LIN {X 0,Y 296.903,Z 465.788,A -85,B 0,C 180,E1 -16297.482,E2 -16297.482} C_VEL
LIN {X 0,Y 297.504,Z 461.29,A -85,B 0,C 180,E1 -16299.52,E2 -16299.52} C_VEL
LIN {X 0,Y 298.387,Z 455.128,A -85,B 0,C 180,E1 -16301.55,E2 -16301.55} C_VEL
LIN {X 0,Y 299.207,Z 450.07,A -85,B 0,C 180,E1 -16302.895,E2 -16302.895} C_VEL
LIN {X 0,Y 300.204,Z 444.009,A -85,B 0,C 180,E1 -16304.232,E2 -16304.232} C_VEL
LIN {X 0,Y 301.376,Z 436.681,A -85,B 0,C 180,E1 -16305.557,E2 -16305.557} C_VEL
LIN {X 0,Y 302.09,Z 430.75,A -85,B 0,C 180,E1 -16306.471,E2 -16306.471} C_VEL
LIN {X 0,Y 302.187,Z 422.359,A -85,B 0,C 180,E1 -16307.6,E2 -16307.6} C_VEL
LIN {X 0,Y 301.805,Z 414.568,A -85,B 0,C 180,E1 -16308.5,E2 -16308.5} C_VEL
LIN {X 0,Y 300.734,Z 405.095,A -85,B 0,C 180,E1 -16309.432,E2 -16309.432} C_VEL
LIN {X 0,Y 298.864,Z 395.139,A -85,B 0,C 180,E1 -16310.262,E2 -16310.262} C_VEL
LIN {X 0,Y 297.662,Z 389.505,A -85,B 0,C 180,E1 -16310.689,E2 -16310.689} C_VEL
LIN {X 0,Y 298.446,Z 382.63,A -85,B 0,C 180,E1 -16315.081,E2 -16315.081} C_VEL
LIN {X 0,Y 299.306,Z 377.058,A -85,B 0,C 180,E1 -16318.776,E2 -16318.776} C_VEL
LIN {X 0,Y 300.359,Z 371.535,A -85,B 0,C 180,E1 -16322.609,E2 -16322.609} C_VEL
LIN {X 0,Y 300.474,Z 369.453,A -85,B 0,C 180,E1 -16324.151,E2 -16324.151} C_VEL
LIN {X 0,Y 300.035,Z 365.619,A -85,B 0,C 180,E1 -16327.21,E2 -16327.21} C_VEL
LIN {X 0,Y 299.34,Z 361.171,A -85,B 0,C 180,E1 -16331.103,E2 -16331.103} C_VEL
LIN {X 0,Y 298.551,Z 357.134,A -85,B 0,C 180,E1 -16335.071,E2 -16335.071} C_VEL
LIN {X 0,Y 298.382,Z 356.135,A -85,B 0,C 180,E1 -16336.22,E2 -16336.22} C_VEL
LIN {X 0,Y 298.411,Z 356.128,A -85,B 0,C 180,E1 -16340.513,E2 -16340.513} C_VEL
LIN {X 0,Y 298.427,Z 356.126,A -85,B 0,C 180,E1 -16343.93,E2 -16343.93} C_VEL
LIN {X 0,Y 298.402,Z 356.129,A -85,B 0,C 180,E1 -16347.984,E2 -16347.984} C_VEL
LIN {X 0,Y 298.467,Z 356.121,A -85,B 0,C 180,E1 -16351.904,E2 -16351.904} C_VEL
LIN {X 0,Y 298.494,Z 356.118,A -85,B 0,C 180,E1 -16354.924,E2 -16354.924} C_VEL
LIN {X 0,Y 298.459,Z 356.121,A -85,B 0,C 180,E1 -16359.315,E2 -16359.315} C_VEL
LIN {X 0,Y 298.546,Z 356.111,A -85,B 0,C 180,E1 -16362.179,E2 -16362.179} C_VEL
LIN {X 0,Y 298.602,Z 356.104,A -85,B 0,C 180,E1 -16364.994,E2 -16364.994} C_VEL
LIN {X 0,Y 298.591,Z 356.104,A -85,B 0,C 180,E1 -16369.145,E2 -16369.145} C_VEL
LIN {X 0,Y 298.72,Z 356.089,A -85,B 0,C 180,E1 -16371.884,E2 -16371.884} C_VEL
LIN {X 0,Y 298.646,Z 356.098,A -85,B 0,C 180,E1 -16374.597,E2 -16374.597} C_VEL
LIN {X 0,Y 298.928,Z 356.059,A -85,B 0,C 180,E1 -16378.652,E2 -16378.652} C_VEL
LIN {X 0,Y 298.928,Z 356.06,A -85,B 0,C 180,E1 -16381.346,E2 -16381.346} C_VEL
LIN {X 0,Y 298.781,Z 356.083,A -85,B 0,C 180,E1 -16386.753,E2 -16386.753} C_VEL
LIN {X 0,Y 298.631,Z 356.1,A -85,B 0,C 180,E1 -16389.481,E2 -16389.481} C_VEL
LIN {X 0,Y 298.544,Z 356.115,A -85,B 0,C 180,E1 -16393.614,E2 -16393.614} C_VEL
LIN {X 0,Y 298.527,Z 356.119,A -85,B 0,C 180,E1 -16395.148,E2 -16395.148} C_VEL
LIN {X 0,Y 298.42,Z 356.43,A -85,B 0,C 180,E1 -16396.414,E2 -16396.414} C_VEL
LIN {X 0,Y 298.385,Z 358.776,A -85,B 0,C 180,E1 -16399.582,E2 -16399.582} C_VEL
LIN {X 0,Y 298.025,Z 362.016,A -85,B 0,C 180,E1 -16403.632,E2 -16403.632} C_VEL
LIN {X 0,Y 297.777,Z 364.531,A -85,B 0,C 180,E1 -16406.641,E2 -16406.641} C_VEL
LIN {X 0,Y 297.563,Z 366.942,A -85,B 0,C 180,E1 -16409.443,E2 -16409.443} C_VEL
LIN {X 0,Y 301.042,Z 378.514,A -85,B 0,C 180,E1 -16410.513,E2 -16410.513} C_VEL
LIN {X 0,Y 303.065,Z 387.21,A -85,B 0,C 180,E1 -16411.449,E2 -16411.449} C_VEL
LIN {X 0,Y 304.331,Z 395.51,A -85,B 0,C 180,E1 -16412.468,E2 -16412.468} C_VEL
LIN {X 0,Y 304.232,Z 400.04,A -85,B 0,C 180,E1 -16413.028,E2 -16413.028} C_VEL
LIN {X 0,Y 303.064,Z 408.255,A -85,B 0,C 180,E1 -16414.191,E2 -16414.191} C_VEL
LIN {X 0,Y 301.948,Z 415.449,A -85,B 0,C 180,E1 -16415.446,E2 -16415.446} C_VEL
LIN {X 0,Y 300.854,Z 422.227,A -85,B 0,C 180,E1 -16416.897,E2 -16416.897} C_VEL
LIN {X 0,Y 299.851,Z 427.76,A -85,B 0,C 180,E1 -16418.344,E2 -16418.344} C_VEL
LIN {X 0,Y 299.089,Z 432.231,A -85,B 0,C 180,E1 -16419.778,E2 -16419.778} C_VEL
LIN {X 0,Y 298.316,Z 436.018,A -85,B 0,C 180,E1 -16421.271,E2 -16421.271} C_VEL
LIN {X 0,Y 297.7,Z 439.323,A -85,B 0,C 180,E1 -16422.957,E2 -16422.957} C_VEL
LIN {X 0,Y 297.154,Z 441.914,A -85,B 0,C 180,E1 -16424.801,E2 -16424.801} C_VEL
LIN {X 0,Y 296.657,Z 443.922,A -85,B 0,C 180,E1 -16427.255,E2 -16427.255} C_VEL
LIN {X 0,Y 296.462,Z 444.243,A -85,B 0,C 180,E1 -16429.338,E2 -16429.338} C_VEL
LIN {X 0,Y 296.511,Z 442.977,A -85,B 0,C 180,E1 -16431.955,E2 -16431.955} C_VEL
LIN {X 0,Y 296.695,Z 441.119,A -85,B 0,C 180,E1 -16433.686,E2 -16433.686} C_VEL
LIN {X 0,Y 297.078,Z 437.521,A -85,B 0,C 180,E1 -16435.89,E2 -16435.89} C_VEL
LIN {X 0,Y 297.534,Z 433.319,A -85,B 0,C 180,E1 -16437.684,E2 -16437.684} C_VEL
LIN {X 0,Y 298.153,Z 427.612,A -85,B 0,C 180,E1 -16439.548,E2 -16439.548} C_VEL
LIN {X 0,Y 298.758,Z 422.641,A -85,B 0,C 180,E1 -16440.866,E2 -16440.866} C_VEL
LIN {X 0,Y 299.406,Z 416.321,A -85,B 0,C 180,E1 -16442.255,E2 -16442.255} C_VEL
LIN {X 0,Y 300.027,Z 410.818,A -85,B 0,C 180,E1 -16443.274,E2 -16443.274} C_VEL
LIN {X 0,Y 300.724,Z 403.711,A -85,B 0,C 180,E1 -16444.382,E2 -16444.382} C_VEL
LIN {X 0,Y 301.459,Z 395.806,A -85,B 0,C 180,E1 -16445.393,E2 -16445.393} C_VEL
LIN {X 0,Y 301.683,Z 390.975,A -85,B 0,C 180,E1 -16445.939,E2 -16445.939} C_VEL
LIN {X 0,Y 300.083,Z 380.873,A -85,B 0,C 180,E1 -16446.933,E2 -16446.933} C_VEL
LIN {X 0,Y 298.191,Z 370.982,A -85,B 0,C 180,E1 -16447.696,E2 -16447.696} C_VEL
LIN {X 0,Y 297.089,Z 365.25,A -85,B 0,C 180,E1 -16448.078,E2 -16448.078} C_VEL
LIN {X 0,Y 297.245,Z 361.276,A -85,B 0,C 180,E1 -16452.098,E2 -16452.098} C_VEL
LIN {X 0,Y 297.576,Z 357.178,A -85,B 0,C 180,E1 -16456.337,E2 -16456.337} C_VEL
LIN {X 0,Y 297.68,Z 356.218,A -85,B 0,C 180,E1 -16457.73,E2 -16457.73} C_VEL
LIN {X 0,Y 298.506,Z 356.113,A -85,B 0,C 180,E1 -16461.877,E2 -16461.877} C_VEL
LIN {X 0,Y 298.621,Z 356.1,A -85,B 0,C 180,E1 -16464.597,E2 -16464.597} C_VEL
LIN {X 0,Y 298.916,Z 356.062,A -85,B 0,C 180,E1 -16468.651,E2 -16468.651} C_VEL
LIN {X 0,Y 298.914,Z 356.061,A -85,B 0,C 180,E1 -16471.346,E2 -16471.346} C_VEL
LIN {X 0,Y 298.789,Z 356.076,A -85,B 0,C 180,E1 -16476.752,E2 -16476.752} C_VEL
LIN {X 0,Y 298.67,Z 356.093,A -85,B 0,C 180,E1 -16479.479,E2 -16479.479} C_VEL
LIN {X 0,Y 298.542,Z 356.11,A -85,B 0,C 180,E1 -16483.614,E2 -16483.614} C_VEL
LIN {X 0,Y 298.537,Z 356.108,A -85,B 0,C 180,E1 -16486.407,E2 -16486.407} C_VEL
LIN {X 0,Y 298.499,Z 356.117,A -85,B 0,C 180,E1 -16489.653,E2 -16489.653} C_VEL
LIN {X 0,Y 298.445,Z 356.124,A -85,B 0,C 180,E1 -16493.597,E2 -16493.597} C_VEL
LIN {X 0,Y 298.476,Z 356.115,A -85,B 0,C 180,E1 -16496.573,E2 -16496.573} C_VEL
LIN {X 0,Y 298.407,Z 356.127,A -85,B 0,C 180,E1 -16499.64,E2 -16499.64} C_VEL
LIN {X 0,Y 298.382,Z 356.128,A -85,B 0,C 180,E1 -16502.799,E2 -16502.799} C_VEL
LIN {X 0,Y 298.458,Z 356.119,A -85,B 0,C 180,E1 -16506.814,E2 -16506.814} C_VEL
LIN {X 0,Y 298.443,Z 356.124,A -85,B 0,C 180,E1 -16511.103,E2 -16511.103} C_VEL
LIN {X 0,Y 298.475,Z 356.12,A -85,B 0,C 180,E1 -16515.061,E2 -16515.061} C_VEL
LIN {X 0,Y 298.443,Z 356.124,A -85,B 0,C 180,E1 -16518.897,E2 -16518.897} C_VEL
LIN {X 0,Y 298.457,Z 356.119,A -85,B 0,C 180,E1 -16523.186,E2 -16523.186} C_VEL
LIN {X 0,Y 298.382,Z 356.129,A -85,B 0,C 180,E1 -16527.2,E2 -16527.2} C_VEL
LIN {X 0,Y 298.418,Z 356.127,A -85,B 0,C 180,E1 -16530.615,E2 -16530.615} C_VEL
LIN {X 0,Y 298.472,Z 356.116,A -85,B 0,C 180,E1 -16533.474,E2 -16533.474} C_VEL
LIN {X 0,Y 298.507,Z 356.115,A -85,B 0,C 180,E1 -16536.66,E2 -16536.66} C_VEL
LIN {X 0,Y 298.554,Z 356.108,A -85,B 0,C 180,E1 -16540.759,E2 -16540.759} C_VEL
LIN {X 0,Y 298.581,Z 356.103,A -85,B 0,C 180,E1 -16544.996,E2 -16544.996} C_VEL
LIN {X 0,Y 298.583,Z 356.102,A -85,B 0,C 180,E1 -16549.148,E2 -16549.148} C_VEL
LIN {X 0,Y 298.747,Z 356.084,A -85,B 0,C 180,E1 -16551.887,E2 -16551.887} C_VEL
LIN {X 0,Y 298.65,Z 356.094,A -85,B 0,C 180,E1 -16554.6,E2 -16554.6} C_VEL
LIN {X 0,Y 298.828,Z 356.071,A -85,B 0,C 180,E1 -16557.415,E2 -16557.415} C_VEL
LIN {X 0,Y 298.194,Z 356.152,A -85,B 0,C 180,E1 -16558.541,E2 -16558.541} C_VEL
LIN {X 0,Y 295.394,Z 356.501,A -85,B 0,C 180,E1 -16560.377,E2 -16560.377} C_VEL
LIN {X 0,Y 292.07,Z 356.914,A -85,B 0,C 180,E1 -16562.628,E2 -16562.628} C_VEL
LIN {X 0,Y 291.651,Z 356.963,A -85,B 0,C 180,E1 -16563.408,E2 -16563.408} C_VEL
LIN {X 0,Y 291.736,Z 356.955,A -85,B 0,C 180,E1 -16566.919,E2 -16566.919} C_VEL
LIN {X 0,Y 291.62,Z 356.974,A -85,B 0,C 180,E1 -16569.713,E2 -16569.713} C_VEL
LIN {X 0,Y 291.514,Z 356.985,A -85,B 0,C 180,E1 -16573.952,E2 -16573.952} C_VEL
LIN {X 0,Y 291.478,Z 356.987,A -85,B 0,C 180,E1 -16576.82,E2 -16576.82} C_VEL
LIN {X 0,Y 291.442,Z 356.992,A -85,B 0,C 180,E1 -16579.877,E2 -16579.877} C_VEL
LIN {X 0,Y 291.392,Z 356.998,A -85,B 0,C 180,E1 -16584.207,E2 -16584.207} C_VEL
LIN {X 0,Y 291.416,Z 357,A -85,B 0,C 180,E1 -16587.273,E2 -16587.273} C_VEL
LIN {X 0,Y 291.331,Z 357.005,A -85,B 0,C 180,E1 -16590.439,E2 -16590.439} C_VEL
LIN {X 0,Y 291.338,Z 357.005,A -85,B 0,C 180,E1 -16593.7,E2 -16593.7} C_VEL
LIN {X 0,Y 291.367,Z 357.004,A -85,B 0,C 180,E1 -16597.255,E2 -16597.255} C_VEL
LIN {X 0,Y 291.327,Z 357.008,A -85,B 0,C 180,E1 -16600.645,E2 -16600.645} C_VEL
LIN {X 0,Y 291.309,Z 357.009,A -85,B 0,C 180,E1 -16604.399,E2 -16604.399} C_VEL
LIN {X 0,Y 291.415,Z 357.077,A -85,B 0,C 180,E1 -16608.646,E2 -16608.646} C_VEL
LIN {X 0,Y 292.375,Z 362.103,A -85,B 0,C 180,E1 -16612.491,E2 -16612.491} C_VEL
LIN {X 0,Y 292.972,Z 366.53,A -85,B 0,C 180,E1 -16615.688,E2 -16615.688} C_VEL
LIN {X 0,Y 292.883,Z 368.616,A -85,B 0,C 180,E1 -16617.126,E2 -16617.126} C_VEL
LIN {X 0,Y 292.227,Z 372.868,A -85,B 0,C 180,E1 -16619.975,E2 -16619.975} C_VEL
LIN {X 0,Y 291.277,Z 379.444,A -85,B 0,C 180,E1 -16624.261,E2 -16624.261} C_VEL
LIN {X 0,Y 290.503,Z 386.389,A -85,B 0,C 180,E1 -16628.724,E2 -16628.724} C_VEL
LIN {X 0,Y 290.108,Z 390.872,A -85,B 0,C 180,E1 -16631.559,E2 -16631.559} C_VEL
LIN {X 0,Y 291.601,Z 403.954,A -85,B 0,C 180,E1 -16632.378,E2 -16632.378} C_VEL
LIN {X 0,Y 292.484,Z 413.89,A -85,B 0,C 180,E1 -16633.243,E2 -16633.243} C_VEL
LIN {X 0,Y 293.002,Z 422.205,A -85,B 0,C 180,E1 -16634.146,E2 -16634.146} C_VEL
LIN {X 0,Y 293.138,Z 429.314,A -85,B 0,C 180,E1 -16635.066,E2 -16635.066} C_VEL
LIN {X 0,Y 292.254,Z 437.158,A -85,B 0,C 180,E1 -16636.265,E2 -16636.265} C_VEL
LIN {X 0,Y 291.523,Z 443.666,A -85,B 0,C 180,E1 -16637.471,E2 -16637.471} C_VEL
LIN {X 0,Y 290.863,Z 449.871,A -85,B 0,C 180,E1 -16638.856,E2 -16638.856} C_VEL
LIN {X 0,Y 290.376,Z 455.026,A -85,B 0,C 180,E1 -16640.248,E2 -16640.248} C_VEL
LIN {X 0,Y 289.995,Z 459.311,A -85,B 0,C 180,E1 -16641.641,E2 -16641.641} C_VEL
LIN {X 0,Y 289.715,Z 462.857,A -85,B 0,C 180,E1 -16643.035,E2 -16643.035} C_VEL
LIN {X 0,Y 289.532,Z 466.528,A -85,B 0,C 180,E1 -16644.896,E2 -16644.896} C_VEL
LIN {X 0,Y 289.575,Z 468.046,A -85,B 0,C 180,E1 -16645.826,E2 -16645.826} C_VEL
LIN {X 0,Y 289.545,Z 469.683,A -85,B 0,C 180,E1 -16647.219,E2 -16647.219} C_VEL
LIN {X 0,Y 289.531,Z 470.791,A -85,B 0,C 180,E1 -16648.611,E2 -16648.611} C_VEL
LIN {X 0,Y 289.582,Z 471.416,A -85,B 0,C 180,E1 -16650.002,E2 -16650.002} C_VEL
LIN {X 0,Y 289.514,Z 471.562,A -85,B 0,C 180,E1 -16651.393,E2 -16651.393} C_VEL
LIN {X 0,Y 289.519,Z 471.172,A -85,B 0,C 180,E1 -16652.785,E2 -16652.785} C_VEL
LIN {X 0,Y 289.505,Z 470.202,A -85,B 0,C 180,E1 -16654.178,E2 -16654.178} C_VEL
LIN {X 0,Y 289.52,Z 468.751,A -85,B 0,C 180,E1 -16655.574,E2 -16655.574} C_VEL
LIN {X 0,Y 289.855,Z 465.607,A -85,B 0,C 180,E1 -16657.665,E2 -16657.665} C_VEL
LIN {X 0,Y 290.472,Z 461.182,A -85,B 0,C 180,E1 -16659.753,E2 -16659.753} C_VEL
LIN {X 0,Y 291.415,Z 455.106,A -85,B 0,C 180,E1 -16661.831,E2 -16661.831} C_VEL
LIN {X 0,Y 292.292,Z 450.124,A -85,B 0,C 180,E1 -16663.206,E2 -16663.206} C_VEL
LIN {X 0,Y 293.333,Z 444.163,A -85,B 0,C 180,E1 -16664.572,E2 -16664.572} C_VEL
LIN {X 0,Y 294.566,Z 436.956,A -85,B 0,C 180,E1 -16665.927,E2 -16665.927} C_VEL
LIN {X 0,Y 295.338,Z 429.614,A -85,B 0,C 180,E1 -16667.089,E2 -16667.089} C_VEL
LIN {X 0,Y 295.352,Z 421.521,A -85,B 0,C 180,E1 -16668.2,E2 -16668.2} C_VEL
LIN {X 0,Y 294.915,Z 413.637,A -85,B 0,C 180,E1 -16669.129,E2 -16669.129} C_VEL
LIN {X 0,Y 293.8,Z 404.622,A -85,B 0,C 180,E1 -16670.045,E2 -16670.045} C_VEL
LIN {X 0,Y 291.838,Z 394.392,A -85,B 0,C 180,E1 -16670.93,E2 -16670.93} C_VEL
LIN {X 0,Y 290.722,Z 389.114,A -85,B 0,C 180,E1 -16671.355,E2 -16671.355} C_VEL
LIN {X 0,Y 291.518,Z 382.516,A -85,B 0,C 180,E1 -16675.72,E2 -16675.72} C_VEL
LIN {X 0,Y 292.266,Z 378.081,A -85,B 0,C 180,E1 -16678.748,E2 -16678.748} C_VEL
LIN {X 0,Y 293.441,Z 372.083,A -85,B 0,C 180,E1 -16683.042,E2 -16683.042} C_VEL
LIN {X 0,Y 293.376,Z 368.98,A -85,B 0,C 180,E1 -16685.462,E2 -16685.462} C_VEL
LIN {X 0,Y 292.834,Z 365.286,A -85,B 0,C 180,E1 -16688.611,E2 -16688.611} C_VEL
LIN {X 0,Y 292.107,Z 361.274,A -85,B 0,C 180,E1 -16692.353,E2 -16692.353} C_VEL
LIN {X 0,Y 291.383,Z 357.005,A -85,B 0,C 180,E1 -16696.931,E2 -16696.931} C_VEL
LIN {X 0,Y 291.361,Z 357.005,A -85,B 0,C 180,E1 -16701.158,E2 -16701.158} C_VEL
LIN {X 0,Y 291.37,Z 357.004,A -85,B 0,C 180,E1 -16704.626,E2 -16704.626} C_VEL
LIN {X 0,Y 291.379,Z 357.004,A -85,B 0,C 180,E1 -16707.95,E2 -16707.95} C_VEL
LIN {X 0,Y 291.386,Z 357.001,A -85,B 0,C 180,E1 -16711.158,E2 -16711.158} C_VEL
LIN {X 0,Y 291.423,Z 356.998,A -85,B 0,C 180,E1 -16714.271,E2 -16714.271} C_VEL
LIN {X 0,Y 291.39,Z 357.001,A -85,B 0,C 180,E1 -16717.299,E2 -16717.299} C_VEL
LIN {X 0,Y 291.467,Z 356.992,A -85,B 0,C 180,E1 -16720.27,E2 -16720.27} C_VEL
LIN {X 0,Y 291.564,Z 356.98,A -85,B 0,C 180,E1 -16724.623,E2 -16724.623} C_VEL
LIN {X 0,Y 291.537,Z 356.983,A -85,B 0,C 180,E1 -16728.879,E2 -16728.879} C_VEL
LIN {X 0,Y 291.671,Z 356.968,A -85,B 0,C 180,E1 -16731.686,E2 -16731.686} C_VEL
LIN {X 0,Y 291.615,Z 356.974,A -85,B 0,C 180,E1 -16734.467,E2 -16734.467} C_VEL
LIN {X 0,Y 291.894,Z 356.935,A -85,B 0,C 180,E1 -16738.619,E2 -16738.619} C_VEL
LIN {X 0,Y 291.894,Z 356.936,A -85,B 0,C 180,E1 -16741.378,E2 -16741.378} C_VEL
LIN {X 0,Y 291.729,Z 356.96,A -85,B 0,C 180,E1 -16746.917,E2 -16746.917} C_VEL
LIN {X 0,Y 291.573,Z 356.98,A -85,B 0,C 180,E1 -16749.712,E2 -16749.712} C_VEL
LIN {X 0,Y 291.504,Z 356.991,A -85,B 0,C 180,E1 -16753.95,E2 -16753.95} C_VEL
LIN {X 0,Y 291.462,Z 357,A -85,B 0,C 180,E1 -16755.38,E2 -16755.38} C_VEL
LIN {X 0,Y 291.416,Z 358.946,A -85,B 0,C 180,E1 -16758.27,E2 -16758.27} C_VEL
LIN {X 0,Y 291.187,Z 361.179,A -85,B 0,C 180,E1 -16761.224,E2 -16761.224} C_VEL
LIN {X 0,Y 290.947,Z 363.568,A -85,B 0,C 180,E1 -16764.244,E2 -16764.244} C_VEL
LIN {X 0,Y 290.611,Z 366.768,A -85,B 0,C 180,E1 -16768.135,E2 -16768.135} C_VEL
LIN {X 0,Y 290.552,Z 367.318,A -85,B 0,C 180,E1 -16768.782,E2 -16768.782} C_VEL
LIN {X 0,Y 293.885,Z 378.073,A -85,B 0,C 180,E1 -16769.815,E2 -16769.815} C_VEL
LIN {X 0,Y 296.191,Z 387.481,A -85,B 0,C 180,E1 -16770.87,E2 -16770.87} C_VEL
LIN {X 0,Y 297.513,Z 395.491,A -85,B 0,C 180,E1 -16771.885,E2 -16771.885} C_VEL
LIN {X 0,Y 297.828,Z 398.291,A -85,B 0,C 180,E1 -16772.266,E2 -16772.266} C_VEL
LIN {X 0,Y 296.435,Z 408.512,A -85,B 0,C 180,E1 -16773.698,E2 -16773.698} C_VEL
LIN {X 0,Y 295.162,Z 416.165,A -85,B 0,C 180,E1 -16775.067,E2 -16775.067} C_VEL
LIN {X 0,Y 294.199,Z 421.9,A -85,B 0,C 180,E1 -16776.313,E2 -16776.313} C_VEL
LIN {X 0,Y 293.202,Z 427.288,A -85,B 0,C 180,E1 -16777.718,E2 -16777.718} C_VEL
LIN {X 0,Y 292.372,Z 431.815,A -85,B 0,C 180,E1 -16779.152,E2 -16779.152} C_VEL
LIN {X 0,Y 291.546,Z 435.598,A -85,B 0,C 180,E1 -16780.604,E2 -16780.604} C_VEL
LIN {X 0,Y 290.764,Z 439.505,A -85,B 0,C 180,E1 -16782.59,E2 -16782.59} C_VEL
LIN {X 0,Y 290.124,Z 442.311,A -85,B 0,C 180,E1 -16784.625,E2 -16784.625} C_VEL
LIN {X 0,Y 289.654,Z 444.03,A -85,B 0,C 180,E1 -16786.708,E2 -16786.708} C_VEL
LIN {X 0,Y 289.396,Z 444.627,A -85,B 0,C 180,E1 -16789.026,E2 -16789.026} C_VEL
LIN {X 0,Y 289.349,Z 443.972,A -85,B 0,C 180,E1 -16791.006,E2 -16791.006} C_VEL
LIN {X 0,Y 289.532,Z 441.999,A -85,B 0,C 180,E1 -16793.225,E2 -16793.225} C_VEL
LIN {X 0,Y 289.721,Z 440.504,A -85,B 0,C 180,E1 -16794.394,E2 -16794.394} C_VEL
LIN {X 0,Y 290.047,Z 437.442,A -85,B 0,C 180,E1 -16796.129,E2 -16796.129} C_VEL
LIN {X 0,Y 290.497,Z 433.412,A -85,B 0,C 180,E1 -16797.857,E2 -16797.857} C_VEL
LIN {X 0,Y 291.053,Z 428.46,A -85,B 0,C 180,E1 -16799.529,E2 -16799.529} C_VEL
LIN {X 0,Y 291.786,Z 422.266,A -85,B 0,C 180,E1 -16801.2,E2 -16801.2} C_VEL
LIN {X 0,Y 292.375,Z 416.814,A -85,B 0,C 180,E1 -16802.418,E2 -16802.418} C_VEL
LIN {X 0,Y 293.146,Z 410.103,A -85,B 0,C 180,E1 -16803.669,E2 -16803.669} C_VEL
LIN {X 0,Y 293.944,Z 402.126,A -85,B 0,C 180,E1 -16804.894,E2 -16804.894} C_VEL
LIN {X 0,Y 294.697,Z 393.776,A -85,B 0,C 180,E1 -16805.933,E2 -16805.933} C_VEL
LIN {X 0,Y 294.368,Z 389.435,A -85,B 0,C 180,E1 -16806.426,E2 -16806.426} C_VEL
LIN {X 0,Y 293.048,Z 381.18,A -85,B 0,C 180,E1 -16807.248,E2 -16807.248} C_VEL
LIN {X 0,Y 291.154,Z 371.388,A -85,B 0,C 180,E1 -16808.027,E2 -16808.027} C_VEL
LIN {X 0,Y 290.004,Z 365.538,A -85,B 0,C 180,E1 -16808.449,E2 -16808.449} C_VEL
LIN {X 0,Y 290.162,Z 362.436,A -85,B 0,C 180,E1 -16811.645,E2 -16811.645} C_VEL
LIN {X 0,Y 290.48,Z 358.307,A -85,B 0,C 180,E1 -16815.997,E2 -16815.997} C_VEL
LIN {X 0,Y 290.577,Z 357.104,A -85,B 0,C 180,E1 -16817.426,E2 -16817.426} C_VEL
LIN {X 0,Y 291.442,Z 356.992,A -85,B 0,C 180,E1 -16821.679,E2 -16821.679} C_VEL
LIN {X 0,Y 291.585,Z 356.978,A -85,B 0,C 180,E1 -16824.466,E2 -16824.466} C_VEL
LIN {X 0,Y 291.882,Z 356.939,A -85,B 0,C 180,E1 -16828.619,E2 -16828.619} C_VEL
LIN {X 0,Y 291.88,Z 356.938,A -85,B 0,C 180,E1 -16831.378,E2 -16831.378} C_VEL
LIN {X 0,Y 291.738,Z 356.955,A -85,B 0,C 180,E1 -16836.916,E2 -16836.916} C_VEL
LIN {X 0,Y 291.619,Z 356.973,A -85,B 0,C 180,E1 -16839.71,E2 -16839.71} C_VEL
LIN {X 0,Y 291.511,Z 356.987,A -85,B 0,C 180,E1 -16843.949,E2 -16843.949} C_VEL
LIN {X 0,Y 291.475,Z 356.987,A -85,B 0,C 180,E1 -16846.817,E2 -16846.817} C_VEL
LIN {X 0,Y 291.438,Z 356.994,A -85,B 0,C 180,E1 -16849.874,E2 -16849.874} C_VEL
LIN {X 0,Y 291.387,Z 356.999,A -85,B 0,C 180,E1 -16854.204,E2 -16854.204} C_VEL
LIN {X 0,Y 291.41,Z 356.999,A -85,B 0,C 180,E1 -16857.271,E2 -16857.271} C_VEL
LIN {X 0,Y 291.324,Z 357.006,A -85,B 0,C 180,E1 -16860.436,E2 -16860.436} C_VEL
LIN {X 0,Y 291.331,Z 357.007,A -85,B 0,C 180,E1 -16863.698,E2 -16863.698} C_VEL
LIN {X 0,Y 291.393,Z 357.002,A -85,B 0,C 180,E1 -16867.261,E2 -16867.261} C_VEL
LIN {X 0,Y 291.393,Z 356.999,A -85,B 0,C 180,E1 -16870.63,E2 -16870.63} C_VEL
LIN {X 0,Y 291.393,Z 356.997,A -85,B 0,C 180,E1 -16874.379,E2 -16874.379} C_VEL
LIN {X 0,Y 291.377,Z 357.001,A -85,B 0,C 180,E1 -16878.39,E2 -16878.39} C_VEL
LIN {X 0,Y 291.374,Z 357.002,A -85,B 0,C 180,E1 -16881.164,E2 -16881.164} C_VEL
LIN {X 0,Y 291.372,Z 357.003,A -85,B 0,C 180,E1 -16884.63,E2 -16884.63} C_VEL
LIN {X 0,Y 291.358,Z 357.002,A -85,B 0,C 180,E1 -16887.951,E2 -16887.951} C_VEL
LIN {X 0,Y 291.369,Z 357.001,A -85,B 0,C 180,E1 -16891.159,E2 -16891.159} C_VEL
LIN {X 0,Y 291.412,Z 356.998,A -85,B 0,C 180,E1 -16894.273,E2 -16894.273} C_VEL
LIN {X 0,Y 291.434,Z 356.992,A -85,B 0,C 180,E1 -16897.306,E2 -16897.306} C_VEL
LIN {X 0,Y 291.501,Z 356.987,A -85,B 0,C 180,E1 -16900.275,E2 -16900.275} C_VEL
LIN {X 0,Y 291.543,Z 356.981,A -85,B 0,C 180,E1 -16904.625,E2 -16904.625} C_VEL
LIN {X 0,Y 291.526,Z 356.981,A -85,B 0,C 180,E1 -16908.882,E2 -16908.882} C_VEL
LIN {X 0,Y 291.697,Z 356.961,A -85,B 0,C 180,E1 -16911.69,E2 -16911.69} C_VEL
LIN {X 0,Y 291.62,Z 356.971,A -85,B 0,C 180,E1 -16914.47,E2 -16914.47} C_VEL
LIN {X 0,Y 291.879,Z 356.938,A -85,B 0,C 180,E1 -16918.622,E2 -16918.622} C_VEL
LIN {X 0,Y 291.881,Z 356.938,A -85,B 0,C 180,E1 -16921.381,E2 -16921.381} C_VEL
LIN {X 0,Y 291.651,Z 356.963,A -85,B 0,C 180,E1 -16923.408,E2 -16923.408} C_VEL
LIN {X 0,Y 290.879,Z 357.062,A -85,B 0,C 180,E1 -16924.56,E2 -16924.56} C_VEL
LIN {X 0,Y 288.083,Z 357.41,A -85,B 0,C 180,E1 -16926.441,E2 -16926.441} C_VEL
LIN {X 0,Y 284.953,Z 357.801,A -85,B 0,C 180,E1 -16928.75,E2 -16928.75} C_VEL
LIN {X 0,Y 284.594,Z 357.845,A -85,B 0,C 180,E1 -16929.546,E2 -16929.546} C_VEL
LIN {X 0,Y 284.473,Z 357.86,A -85,B 0,C 180,E1 -16934.304,E2 -16934.304} C_VEL
LIN {X 0,Y 284.417,Z 357.869,A -85,B 0,C 180,E1 -16937.25,E2 -16937.25} C_VEL
LIN {X 0,Y 284.371,Z 357.872,A -85,B 0,C 180,E1 -16940.244,E2 -16940.244} C_VEL
LIN {X 0,Y 284.362,Z 357.875,A -85,B 0,C 180,E1 -16943.877,E2 -16943.877} C_VEL
LIN {X 0,Y 284.39,Z 357.874,A -85,B 0,C 180,E1 -16947.176,E2 -16947.176} C_VEL
LIN {X 0,Y 284.289,Z 357.887,A -85,B 0,C 180,E1 -16951.276,E2 -16951.276} C_VEL
LIN {X 0,Y 284.335,Z 357.879,A -85,B 0,C 180,E1 -16955.35,E2 -16955.35} C_VEL
LIN {X 0,Y 284.303,Z 357.88,A -85,B 0,C 180,E1 -16958.172,E2 -16958.172} C_VEL
LIN {X 0,Y 284.264,Z 357.886,A -85,B 0,C 180,E1 -16962.127,E2 -16962.127} C_VEL
LIN {X 0,Y 284.281,Z 357.884,A -85,B 0,C 180,E1 -16966.197,E2 -16966.197} C_VEL
LIN {X 0,Y 284.358,Z 358.006,A -85,B 0,C 180,E1 -16968.495,E2 -16968.495} C_VEL
LIN {X 0,Y 285.216,Z 362.531,A -85,B 0,C 180,E1 -16972.048,E2 -16972.048} C_VEL
LIN {X 0,Y 285.935,Z 367.27,A -85,B 0,C 180,E1 -16975.578,E2 -16975.578} C_VEL
LIN {X 0,Y 285.807,Z 369.643,A -85,B 0,C 180,E1 -16977.252,E2 -16977.252} C_VEL
LIN {X 0,Y 284.854,Z 375.483,A -85,B 0,C 180,E1 -16981.244,E2 -16981.244} C_VEL
LIN {X 0,Y 283.99,Z 381.297,A -85,B 0,C 180,E1 -16985.123,E2 -16985.123} C_VEL
LIN {X 0,Y 283.387,Z 387.087,A -85,B 0,C 180,E1 -16988.927,E2 -16988.927} C_VEL
LIN {X 0,Y 283.079,Z 390.547,A -85,B 0,C 180,E1 -16991.173,E2 -16991.173} C_VEL
LIN {X 0,Y 284.541,Z 403.382,A -85,B 0,C 180,E1 -16992.019,E2 -16992.019} C_VEL
LIN {X 0,Y 285.359,Z 412.423,A -85,B 0,C 180,E1 -16992.812,E2 -16992.812} C_VEL
LIN {X 0,Y 285.914,Z 421.408,A -85,B 0,C 180,E1 -16993.796,E2 -16993.796} C_VEL
LIN {X 0,Y 286.114,Z 429.484,A -85,B 0,C 180,E1 -16994.873,E2 -16994.873} C_VEL
LIN {X 0,Y 285.214,Z 437.244,A -85,B 0,C 180,E1 -16996.101,E2 -16996.101} C_VEL
LIN {X 0,Y 284.374,Z 444.536,A -85,B 0,C 180,E1 -16997.513,E2 -16997.513} C_VEL
LIN {X 0,Y 283.586,Z 451.945,A -85,B 0,C 180,E1 -16999.29,E2 -16999.29} C_VEL
LIN {X 0,Y 283.032,Z 457.734,A -85,B 0,C 180,E1 -17001.074,E2 -17001.074} C_VEL
LIN {X 0,Y 282.662,Z 462.301,A -85,B 0,C 180,E1 -17002.861,E2 -17002.861} C_VEL
LIN {X 0,Y 282.439,Z 466.367,A -85,B 0,C 180,E1 -17004.98,E2 -17004.98} C_VEL
LIN {X 0,Y 282.489,Z 467.559,A -85,B 0,C 180,E1 -17005.722,E2 -17005.722} C_VEL
LIN {X 0,Y 282.473,Z 469.231,A -85,B 0,C 180,E1 -17007.15,E2 -17007.15} C_VEL
LIN {X 0,Y 282.449,Z 470.386,A -85,B 0,C 180,E1 -17008.576,E2 -17008.576} C_VEL
LIN {X 0,Y 282.495,Z 471.056,A -85,B 0,C 180,E1 -17010.002,E2 -17010.002} C_VEL
LIN {X 0,Y 282.433,Z 471.245,A -85,B 0,C 180,E1 -17011.428,E2 -17011.428} C_VEL
LIN {X 0,Y 282.445,Z 470.86,A -85,B 0,C 180,E1 -17012.854,E2 -17012.854} C_VEL
LIN {X 0,Y 282.422,Z 468.781,A -85,B 0,C 180,E1 -17015.497,E2 -17015.497} C_VEL
LIN {X 0,Y 282.793,Z 465.431,A -85,B 0,C 180,E1 -17017.858,E2 -17017.858} C_VEL
LIN {X 0,Y 283.456,Z 461.083,A -85,B 0,C 180,E1 -17019.997,E2 -17019.997} C_VEL
LIN {X 0,Y 284.466,Z 455.139,A -85,B 0,C 180,E1 -17022.124,E2 -17022.124} C_VEL
LIN {X 0,Y 285.589,Z 448.814,A -85,B 0,C 180,E1 -17023.884,E2 -17023.884} C_VEL
LIN {X 0,Y 286.73,Z 442.665,A -85,B 0,C 180,E1 -17025.279,E2 -17025.279} C_VEL
LIN {X 0,Y 287.91,Z 436.25,A -85,B 0,C 180,E1 -17026.487,E2 -17026.487} C_VEL
LIN {X 0,Y 288.546,Z 430.243,A -85,B 0,C 180,E1 -17027.475,E2 -17027.475} C_VEL
LIN {X 0,Y 288.615,Z 422.127,A -85,B 0,C 180,E1 -17028.641,E2 -17028.641} C_VEL
LIN {X 0,Y 288.211,Z 414.483,A -85,B 0,C 180,E1 -17029.592,E2 -17029.592} C_VEL
LIN {X 0,Y 287.182,Z 405.595,A -85,B 0,C 180,E1 -17030.554,E2 -17030.554} C_VEL
LIN {X 0,Y 285.362,Z 395.938,A -85,B 0,C 180,E1 -17031.455,E2 -17031.455} C_VEL
LIN {X 0,Y 283.763,Z 388.785,A -85,B 0,C 180,E1 -17032.049,E2 -17032.049} C_VEL
LIN {X 0,Y 284.604,Z 382.426,A -85,B 0,C 180,E1 -17036.393,E2 -17036.393} C_VEL
LIN {X 0,Y 285.676,Z 376.57,A -85,B 0,C 180,E1 -17040.564,E2 -17040.564} C_VEL
LIN {X 0,Y 286.543,Z 372.636,A -85,B 0,C 180,E1 -17043.496,E2 -17043.496} C_VEL
LIN {X 0,Y 286.115,Z 368.434,A -85,B 0,C 180,E1 -17047.001,E2 -17047.001} C_VEL
LIN {X 0,Y 285.563,Z 364.845,A -85,B 0,C 180,E1 -17050.274,E2 -17050.274} C_VEL
LIN {X 0,Y 284.819,Z 360.852,A -85,B 0,C 180,E1 -17054.308,E2 -17054.308} C_VEL
LIN {X 0,Y 284.305,Z 357.886,A -85,B 0,C 180,E1 -17057.773,E2 -17057.773} C_VEL
LIN {X 0,Y 284.32,Z 357.883,A -85,B 0,C 180,E1 -17061.831,E2 -17061.831} C_VEL
LIN {X 0,Y 284.317,Z 357.883,A -85,B 0,C 180,E1 -17065.351,E2 -17065.351} C_VEL
LIN {X 0,Y 284.302,Z 357.885,A -85,B 0,C 180,E1 -17068.725,E2 -17068.725} C_VEL
LIN {X 0,Y 284.404,Z 357.872,A -85,B 0,C 180,E1 -17072.827,E2 -17072.827} C_VEL
LIN {X 0,Y 284.375,Z 357.875,A -85,B 0,C 180,E1 -17076.707,E2 -17076.707} C_VEL
LIN {X 0,Y 284.412,Z 357.87,A -85,B 0,C 180,E1 -17081.261,E2 -17081.261} C_VEL
LIN {X 0,Y 284.501,Z 357.859,A -85,B 0,C 180,E1 -17084.458,E2 -17084.458} C_VEL
LIN {X 0,Y 284.49,Z 357.861,A -85,B 0,C 180,E1 -17088.6,E2 -17088.6} C_VEL
LIN {X 0,Y 284.626,Z 357.845,A -85,B 0,C 180,E1 -17091.479,E2 -17091.479} C_VEL
LIN {X 0,Y 284.585,Z 357.851,A -85,B 0,C 180,E1 -17094.33,E2 -17094.33} C_VEL
LIN {X 0,Y 284.86,Z 357.811,A -85,B 0,C 180,E1 -17098.585,E2 -17098.585} C_VEL
LIN {X 0,Y 284.861,Z 357.812,A -85,B 0,C 180,E1 -17101.412,E2 -17101.412} C_VEL
LIN {X 0,Y 284.679,Z 357.838,A -85,B 0,C 180,E1 -17107.089,E2 -17107.089} C_VEL
LIN {X 0,Y 284.519,Z 357.859,A -85,B 0,C 180,E1 -17109.955,E2 -17109.955} C_VEL
LIN {X 0,Y 284.451,Z 357.871,A -85,B 0,C 180,E1 -17114.303,E2 -17114.303} C_VEL
LIN {X 0,Y 284.446,Z 358.391,A -85,B 0,C 180,E1 -17115.769,E2 -17115.769} C_VEL
LIN {X 0,Y 284.306,Z 361.404,A -85,B 0,C 180,E1 -17120.053,E2 -17120.053} C_VEL
LIN {X 0,Y 283.972,Z 364.195,A -85,B 0,C 180,E1 -17123.69,E2 -17123.69} C_VEL
LIN {X 0,Y 283.621,Z 367.44,A -85,B 0,C 180,E1 -17127.751,E2 -17127.751} C_VEL
LIN {X 0,Y 283.599,Z 367.847,A -85,B 0,C 180,E1 -17128.087,E2 -17128.087} C_VEL
LIN {X 0,Y 287.32,Z 379.582,A -85,B 0,C 180,E1 -17129.287,E2 -17129.287} C_VEL
LIN {X 0,Y 289.451,Z 388.306,A -85,B 0,C 180,E1 -17130.319,E2 -17130.319} C_VEL
LIN {X 0,Y 290.739,Z 395.754,A -85,B 0,C 180,E1 -17131.311,E2 -17131.311} C_VEL
LIN {X 0,Y 290.968,Z 401.422,A -85,B 0,C 180,E1 -17132.097,E2 -17132.097} C_VEL
LIN {X 0,Y 289.562,Z 410.212,A -85,B 0,C 180,E1 -17133.43,E2 -17133.43} C_VEL
LIN {X 0,Y 288.347,Z 417.223,A -85,B 0,C 180,E1 -17134.745,E2 -17134.745} C_VEL
LIN {X 0,Y 287.218,Z 423.361,A -85,B 0,C 180,E1 -17136.147,E2 -17136.147} C_VEL
LIN {X 0,Y 286.21,Z 428.471,A -85,B 0,C 180,E1 -17137.559,E2 -17137.559} C_VEL
LIN {X 0,Y 285.335,Z 432.971,A -85,B 0,C 180,E1 -17139.075,E2 -17139.075} C_VEL
LIN {X 0,Y 284.49,Z 436.591,A -85,B 0,C 180,E1 -17140.566,E2 -17140.566} C_VEL
LIN {X 0,Y 283.886,Z 439.452,A -85,B 0,C 180,E1 -17142.037,E2 -17142.037} C_VEL
LIN {X 0,Y 283.213,Z 442.252,A -85,B 0,C 180,E1 -17144.011,E2 -17144.011} C_VEL
LIN {X 0,Y 282.683,Z 444.127,A -85,B 0,C 180,E1 -17146.134,E2 -17146.134} C_VEL
LIN {X 0,Y 282.349,Z 444.91,A -85,B 0,C 180,E1 -17148.306,E2 -17148.306} C_VEL
LIN {X 0,Y 282.268,Z 444.545,A -85,B 0,C 180,E1 -17150.517,E2 -17150.517} C_VEL
LIN {X 0,Y 282.468,Z 442.184,A -85,B 0,C 180,E1 -17153.333,E2 -17153.333} C_VEL
LIN {X 0,Y 282.73,Z 439.639,A -85,B 0,C 180,E1 -17155.128,E2 -17155.128} C_VEL
LIN {X 0,Y 283.162,Z 436.204,A -85,B 0,C 180,E1 -17156.903,E2 -17156.903} C_VEL
LIN {X 0,Y 283.762,Z 430.876,A -85,B 0,C 180,E1 -17159.001,E2 -17159.001} C_VEL
LIN {X 0,Y 284.505,Z 424.924,A -85,B 0,C 180,E1 -17160.797,E2 -17160.797} C_VEL
LIN {X 0,Y 285.34,Z 417.34,A -85,B 0,C 180,E1 -17162.582,E2 -17162.582} C_VEL
LIN {X 0,Y 286.171,Z 410.314,A -85,B 0,C 180,E1 -17163.924,E2 -17163.924} C_VEL
LIN {X 0,Y 286.951,Z 402.735,A -85,B 0,C 180,E1 -17165.118,E2 -17165.118} C_VEL
LIN {X 0,Y 287.639,Z 395.714,A -85,B 0,C 180,E1 -17166.032,E2 -17166.032} C_VEL
LIN {X 0,Y 287.513,Z 391.058,A -85,B 0,C 180,E1 -17166.594,E2 -17166.594} C_VEL
LIN {X 0,Y 285.924,Z 381.236,A -85,B 0,C 180,E1 -17167.603,E2 -17167.603} C_VEL
LIN {X 0,Y 284.031,Z 371.423,A -85,B 0,C 180,E1 -17168.402,E2 -17168.402} C_VEL
LIN {X 0,Y 282.941,Z 365.87,A -85,B 0,C 180,E1 -17168.792,E2 -17168.792} C_VEL
LIN {X 0,Y 283.134,Z 362.185,A -85,B 0,C 180,E1 -17172.669,E2 -17172.669} C_VEL
LIN {X 0,Y 283.401,Z 359.428,A -85,B 0,C 180,E1 -17175.64,E2 -17175.64} C_VEL
LIN {X 0,Y 283.563,Z 357.977,A -85,B 0,C 180,E1 -17177.473,E2 -17177.473} C_VEL
LIN {X 0,Y 284.344,Z 357.876,A -85,B 0,C 180,E1 -17181.47,E2 -17181.47} C_VEL
LIN {X 0,Y 284.548,Z 357.856,A -85,B 0,C 180,E1 -17184.328,E2 -17184.328} C_VEL
LIN {X 0,Y 284.848,Z 357.815,A -85,B 0,C 180,E1 -17188.584,E2 -17188.584} C_VEL
LIN {X 0,Y 284.846,Z 357.814,A -85,B 0,C 180,E1 -17191.412,E2 -17191.412} C_VEL
LIN {X 0,Y 284.69,Z 357.833,A -85,B 0,C 180,E1 -17197.088,E2 -17197.088} C_VEL
LIN {X 0,Y 284.556,Z 357.853,A -85,B 0,C 180,E1 -17199.954,E2 -17199.954} C_VEL
LIN {X 0,Y 284.471,Z 357.861,A -85,B 0,C 180,E1 -17204.301,E2 -17204.301} C_VEL
LIN {X 0,Y 284.413,Z 357.869,A -85,B 0,C 180,E1 -17207.247,E2 -17207.247} C_VEL
LIN {X 0,Y 284.368,Z 357.873,A -85,B 0,C 180,E1 -17210.241,E2 -17210.241} C_VEL
LIN {X 0,Y 284.356,Z 357.877,A -85,B 0,C 180,E1 -17213.874,E2 -17213.874} C_VEL
LIN {X 0,Y 284.384,Z 357.873,A -85,B 0,C 180,E1 -17217.173,E2 -17217.173} C_VEL
LIN {X 0,Y 284.282,Z 357.887,A -85,B 0,C 180,E1 -17221.273,E2 -17221.273} C_VEL
LIN {X 0,Y 284.349,Z 357.878,A -85,B 0,C 180,E1 -17225.354,E2 -17225.354} C_VEL
LIN {X 0,Y 284.325,Z 357.878,A -85,B 0,C 180,E1 -17228.164,E2 -17228.164} C_VEL
LIN {X 0,Y 284.331,Z 357.877,A -85,B 0,C 180,E1 -17232.141,E2 -17232.141} C_VEL
LIN {X 0,Y 284.339,Z 357.876,A -85,B 0,C 180,E1 -17236.208,E2 -17236.208} C_VEL
LIN {X 0,Y 284.337,Z 357.877,A -85,B 0,C 180,E1 -17240.013,E2 -17240.013} C_VEL
LIN {X 0,Y 284.342,Z 357.875,A -85,B 0,C 180,E1 -17243.618,E2 -17243.618} C_VEL
LIN {X 0,Y 284.294,Z 357.884,A -85,B 0,C 180,E1 -17247.19,E2 -17247.19} C_VEL
LIN {X 0,Y 284.345,Z 357.878,A -85,B 0,C 180,E1 -17250.376,E2 -17250.376} C_VEL
LIN {X 0,Y 284.368,Z 357.873,A -85,B 0,C 180,E1 -17253.587,E2 -17253.587} C_VEL
LIN {X 0,Y 284.39,Z 357.873,A -85,B 0,C 180,E1 -17256.711,E2 -17256.711} C_VEL
LIN {X 0,Y 284.423,Z 357.866,A -85,B 0,C 180,E1 -17259.872,E2 -17259.872} C_VEL
LIN {X 0,Y 284.48,Z 357.863,A -85,B 0,C 180,E1 -17264.46,E2 -17264.46} C_VEL
LIN {X 0,Y 284.478,Z 357.861,A -85,B 0,C 180,E1 -17268.603,E2 -17268.603} C_VEL
LIN {X 0,Y 284.647,Z 357.838,A -85,B 0,C 180,E1 -17271.482,E2 -17271.482} C_VEL
LIN {X 0,Y 284.591,Z 357.847,A -85,B 0,C 180,E1 -17274.333,E2 -17274.333} C_VEL
LIN {X 0,Y 284.845,Z 357.814,A -85,B 0,C 180,E1 -17278.588,E2 -17278.588} C_VEL
LIN {X 0,Y 284.847,Z 357.814,A -85,B 0,C 180,E1 -17281.415,E2 -17281.415} C_VEL
LIN {X 0,Y 284.689,Z 357.833,A -85,B 0,C 180,E1 -17287.092,E2 -17287.092} C_VEL
LIN {X 0,Y 284.594,Z 357.845,A -85,B 0,C 180,E1 -17289.546,E2 -17289.546} C_VEL
LIN {X 0,Y 283.857,Z 357.941,A -85,B 0,C 180,E1 -17290.726,E2 -17290.726} C_VEL
LIN {X 0,Y 281.012,Z 358.302,A -85,B 0,C 180,E1 -17292.648,E2 -17292.648} C_VEL
LIN {X 0,Y 278.612,Z 358.601,A -85,B 0,C 180,E1 -17294.208,E2 -17294.208} C_VEL
LIN {X 0,Y 277.538,Z 358.729,A -85,B 0,C 180,E1 -17295.416,E2 -17295.416} C_VEL
LIN {X 0,Y 277.425,Z 358.741,A -85,B 0,C 180,E1 -17295.826,E2 -17295.826} C_VEL
LIN {X 0,Y 277.337,Z 358.747,A -85,B 0,C 180,E1 -17300.352,E2 -17300.352} C_VEL
LIN {X 0,Y 277.312,Z 358.752,A -85,B 0,C 180,E1 -17304.172,E2 -17304.172} C_VEL
LIN {X 0,Y 277.319,Z 358.753,A -85,B 0,C 180,E1 -17307.507,E2 -17307.507} C_VEL
LIN {X 0,Y 277.265,Z 358.757,A -85,B 0,C 180,E1 -17310.483,E2 -17310.483} C_VEL
LIN {X 0,Y 277.241,Z 358.761,A -85,B 0,C 180,E1 -17313.898,E2 -17313.898} C_VEL
LIN {X 0,Y 277.259,Z 358.759,A -85,B 0,C 180,E1 -17317.472,E2 -17317.472} C_VEL
LIN {X 0,Y 277.205,Z 358.768,A -85,B 0,C 180,E1 -17321.239,E2 -17321.239} C_VEL
LIN {X 0,Y 277.218,Z 358.765,A -85,B 0,C 180,E1 -17325.224,E2 -17325.224} C_VEL
LIN {X 0,Y 277.303,Z 358.886,A -85,B 0,C 180,E1 -17328.299,E2 -17328.299} C_VEL
LIN {X 0,Y 278.093,Z 362.936,A -85,B 0,C 180,E1 -17331.578,E2 -17331.578} C_VEL
LIN {X 0,Y 278.747,Z 366.801,A -85,B 0,C 180,E1 -17334.56,E2 -17334.56} C_VEL
LIN {X 0,Y 278.883,Z 369.188,A -85,B 0,C 180,E1 -17336.332,E2 -17336.332} C_VEL
LIN {X 0,Y 278.186,Z 373.861,A -85,B 0,C 180,E1 -17339.653,E2 -17339.653} C_VEL
LIN {X 0,Y 277.202,Z 379.69,A -85,B 0,C 180,E1 -17343.663,E2 -17343.663} C_VEL
LIN {X 0,Y 276.377,Z 386.599,A -85,B 0,C 180,E1 -17348.365,E2 -17348.365} C_VEL
LIN {X 0,Y 276.012,Z 390.254,A -85,B 0,C 180,E1 -17350.817,E2 -17350.817} C_VEL
LIN {X 0,Y 277.477,Z 402.771,A -85,B 0,C 180,E1 -17351.64,E2 -17351.64} C_VEL
LIN {X 0,Y 278.324,Z 412.566,A -85,B 0,C 180,E1 -17352.526,E2 -17352.526} C_VEL
LIN {X 0,Y 278.836,Z 420.717,A -85,B 0,C 180,E1 -17353.442,E2 -17353.442} C_VEL
LIN {X 0,Y 279.114,Z 428.414,A -85,B 0,C 180,E1 -17354.484,E2 -17354.484} C_VEL
LIN {X 0,Y 278.335,Z 436.316,A -85,B 0,C 180,E1 -17355.75,E2 -17355.75} C_VEL
LIN {X 0,Y 277.416,Z 443.7,A -85,B 0,C 180,E1 -17357.195,E2 -17357.195} C_VEL
LIN {X 0,Y 276.598,Z 451.214,A -85,B 0,C 180,E1 -17359.016,E2 -17359.016} C_VEL
LIN {X 0,Y 275.918,Z 458.081,A -85,B 0,C 180,E1 -17361.211,E2 -17361.211} C_VEL
LIN {X 0,Y 275.502,Z 463.267,A -85,B 0,C 180,E1 -17363.41,E2 -17363.41} C_VEL
LIN {X 0,Y 275.384,Z 467.058,A -85,B 0,C 180,E1 -17365.611,E2 -17365.611} C_VEL
LIN {X 0,Y 275.401,Z 468.778,A -85,B 0,C 180,E1 -17367.076,E2 -17367.076} C_VEL
LIN {X 0,Y 275.37,Z 469.98,A -85,B 0,C 180,E1 -17368.539,E2 -17368.539} C_VEL
LIN {X 0,Y 275.41,Z 470.696,A -85,B 0,C 180,E1 -17370.002,E2 -17370.002} C_VEL
LIN {X 0,Y 275.354,Z 470.918,A -85,B 0,C 180,E1 -17371.464,E2 -17371.464} C_VEL
LIN {X 0,Y 275.371,Z 470.546,A -85,B 0,C 180,E1 -17372.928,E2 -17372.928} C_VEL
LIN {X 0,Y 275.345,Z 468.778,A -85,B 0,C 180,E1 -17375.461,E2 -17375.461} C_VEL
LIN {X 0,Y 275.753,Z 465.28,A -85,B 0,C 180,E1 -17378.06,E2 -17378.06} C_VEL
LIN {X 0,Y 276.183,Z 462.546,A -85,B 0,C 180,E1 -17379.523,E2 -17379.523} C_VEL
LIN {X 0,Y 277.107,Z 457.257,A -85,B 0,C 180,E1 -17381.708,E2 -17381.708} C_VEL
LIN {X 0,Y 278.479,Z 450.347,A -85,B 0,C 180,E1 -17383.874,E2 -17383.874} C_VEL
LIN {X 0,Y 279.902,Z 442.865,A -85,B 0,C 180,E1 -17385.661,E2 -17385.661} C_VEL
LIN {X 0,Y 281.261,Z 435.55,A -85,B 0,C 180,E1 -17387.076,E2 -17387.076} C_VEL
LIN {X 0,Y 281.807,Z 429.55,A -85,B 0,C 180,E1 -17388.09,E2 -17388.09} C_VEL
LIN {X 0,Y 281.848,Z 421.402,A -85,B 0,C 180,E1 -17389.294,E2 -17389.294} C_VEL
LIN {X 0,Y 281.418,Z 413.756,A -85,B 0,C 180,E1 -17390.276,E2 -17390.276} C_VEL
LIN {X 0,Y 280.378,Z 405.428,A -85,B 0,C 180,E1 -17391.214,E2 -17391.214} C_VEL
LIN {X 0,Y 278.648,Z 396.214,A -85,B 0,C 180,E1 -17392.114,E2 -17392.114} C_VEL
LIN {X 0,Y 276.806,Z 388.432,A -85,B 0,C 180,E1 -17392.782,E2 -17392.782} C_VEL
LIN {X 0,Y 277.722,Z 382.341,A -85,B 0,C 180,E1 -17397.099,E2 -17397.099} C_VEL
LIN {X 0,Y 278.757,Z 377.048,A -85,B 0,C 180,E1 -17400.994,E2 -17400.994} C_VEL
LIN {X 0,Y 279.523,Z 373.264,A -85,B 0,C 180,E1 -17403.929,E2 -17403.929} C_VEL
LIN {X 0,Y 279.103,Z 369.501,A -85,B 0,C 180,E1 -17407.183,E2 -17407.183} C_VEL
LIN {X 0,Y 278.449,Z 365.45,A -85,B 0,C 180,E1 -17411.015,E2 -17411.015} C_VEL
LIN {X 0,Y 277.723,Z 361.586,A -85,B 0,C 180,E1 -17415.12,E2 -17415.12} C_VEL
LIN {X 0,Y 277.233,Z 358.766,A -85,B 0,C 180,E1 -17418.577,E2 -17418.577} C_VEL
LIN {X 0,Y 277.276,Z 358.76,A -85,B 0,C 180,E1 -17422.531,E2 -17422.531} C_VEL
LIN {X 0,Y 277.256,Z 358.762,A -85,B 0,C 180,E1 -17426.104,E2 -17426.104} C_VEL
LIN {X 0,Y 277.27,Z 358.76,A -85,B 0,C 180,E1 -17429.538,E2 -17429.538} C_VEL
LIN {X 0,Y 277.366,Z 358.749,A -85,B 0,C 180,E1 -17432.864,E2 -17432.864} C_VEL
LIN {X 0,Y 277.337,Z 358.753,A -85,B 0,C 180,E1 -17436.079,E2 -17436.079} C_VEL
LIN {X 0,Y 277.354,Z 358.75,A -85,B 0,C 180,E1 -17440.766,E2 -17440.766} C_VEL
LIN {X 0,Y 277.443,Z 358.739,A -85,B 0,C 180,E1 -17445.325,E2 -17445.325} C_VEL
LIN {X 0,Y 277.465,Z 358.737,A -85,B 0,C 180,E1 -17449.786,E2 -17449.786} C_VEL
LIN {X 0,Y 277.618,Z 358.717,A -85,B 0,C 180,E1 -17452.727,E2 -17452.727} C_VEL
LIN {X 0,Y 277.826,Z 358.687,A -85,B 0,C 180,E1 -17458.549,E2 -17458.549} C_VEL
LIN {X 0,Y 277.827,Z 358.688,A -85,B 0,C 180,E1 -17461.448,E2 -17461.448} C_VEL
LIN {X 0,Y 277.634,Z 358.715,A -85,B 0,C 180,E1 -17467.27,E2 -17467.27} C_VEL
LIN {X 0,Y 277.463,Z 358.737,A -85,B 0,C 180,E1 -17470.211,E2 -17470.211} C_VEL
LIN {X 0,Y 277.406,Z 358.746,A -85,B 0,C 180,E1 -17473.178,E2 -17473.178} C_VEL
LIN {X 0,Y 277.4,Z 358.938,A -85,B 0,C 180,E1 -17474.674,E2 -17474.674} C_VEL
LIN {X 0,Y 277.376,Z 360.921,A -85,B 0,C 180,E1 -17477.699,E2 -17477.699} C_VEL
LIN {X 0,Y 277.191,Z 363.105,A -85,B 0,C 180,E1 -17480.789,E2 -17480.789} C_VEL
LIN {X 0,Y 276.909,Z 365.487,A -85,B 0,C 180,E1 -17483.977,E2 -17483.977} C_VEL
LIN {X 0,Y 276.603,Z 368.074,A -85,B 0,C 180,E1 -17487.298,E2 -17487.298} C_VEL
LIN {X 0,Y 280.472,Z 380.092,A -85,B 0,C 180,E1 -17488.613,E2 -17488.613} C_VEL
LIN {X 0,Y 282.54,Z 388.161,A -85,B 0,C 180,E1 -17489.606,E2 -17489.606} C_VEL
LIN {X 0,Y 283.964,Z 396.059,A -85,B 0,C 180,E1 -17490.692,E2 -17490.692} C_VEL
LIN {X 0,Y 284.452,Z 401.186,A -85,B 0,C 180,E1 -17491.443,E2 -17491.443} C_VEL
LIN {X 0,Y 282.977,Z 410.577,A -85,B 0,C 180,E1 -17492.905,E2 -17492.905} C_VEL
LIN {X 0,Y 281.767,Z 417.062,A -85,B 0,C 180,E1 -17494.137,E2 -17494.137} C_VEL
LIN {X 0,Y 280.619,Z 423.047,A -85,B 0,C 180,E1 -17495.514,E2 -17495.514} C_VEL
LIN {X 0,Y 279.401,Z 428.824,A -85,B 0,C 180,E1 -17497.132,E2 -17497.132} C_VEL
LIN {X 0,Y 278.533,Z 432.944,A -85,B 0,C 180,E1 -17498.535,E2 -17498.535} C_VEL
LIN {X 0,Y 277.411,Z 437.599,A -85,B 0,C 180,E1 -17500.531,E2 -17500.531} C_VEL
LIN {X 0,Y 276.596,Z 441.057,A -85,B 0,C 180,E1 -17502.533,E2 -17502.533} C_VEL
LIN {X 0,Y 275.977,Z 443.427,A -85,B 0,C 180,E1 -17504.515,E2 -17504.515} C_VEL
LIN {X 0,Y 275.543,Z 444.818,A -85,B 0,C 180,E1 -17506.474,E2 -17506.474} C_VEL
LIN {X 0,Y 275.249,Z 445.301,A -85,B 0,C 180,E1 -17508.403,E2 -17508.403} C_VEL
LIN {X 0,Y 275.184,Z 444.915,A -85,B 0,C 180,E1 -17510.319,E2 -17510.319} C_VEL
LIN {X 0,Y 275.278,Z 443.603,A -85,B 0,C 180,E1 -17512.318,E2 -17512.318} C_VEL
LIN {X 0,Y 275.593,Z 440.711,A -85,B 0,C 180,E1 -17514.687,E2 -17514.687} C_VEL
LIN {X 0,Y 275.968,Z 437.376,A -85,B 0,C 180,E1 -17516.571,E2 -17516.571} C_VEL
LIN {X 0,Y 276.409,Z 433.772,A -85,B 0,C 180,E1 -17518.155,E2 -17518.155} C_VEL
LIN {X 0,Y 277.064,Z 428.303,A -85,B 0,C 180,E1 -17520.049,E2 -17520.049} C_VEL
LIN {X 0,Y 277.711,Z 423.094,A -85,B 0,C 180,E1 -17521.511,E2 -17521.511} C_VEL
LIN {X 0,Y 278.441,Z 416.791,A -85,B 0,C 180,E1 -17522.976,E2 -17522.976} C_VEL
LIN {X 0,Y 279.261,Z 410.064,A -85,B 0,C 180,E1 -17524.269,E2 -17524.269} C_VEL
LIN {X 0,Y 280.135,Z 402.001,A -85,B 0,C 180,E1 -17525.545,E2 -17525.545} C_VEL
LIN {X 0,Y 280.798,Z 393.925,A -85,B 0,C 180,E1 -17526.587,E2 -17526.587} C_VEL
LIN {X 0,Y 279.138,Z 383.044,A -85,B 0,C 180,E1 -17527.809,E2 -17527.809} C_VEL
LIN {X 0,Y 277.132,Z 372.324,A -85,B 0,C 180,E1 -17528.716,E2 -17528.716} C_VEL
LIN {X 0,Y 275.858,Z 366.192,A -85,B 0,C 180,E1 -17529.154,E2 -17529.154} C_VEL
LIN {X 0,Y 276.024,Z 363.345,A -85,B 0,C 180,E1 -17532.208,E2 -17532.208} C_VEL
LIN {X 0,Y 276.32,Z 360.551,A -85,B 0,C 180,E1 -17535.264,E2 -17535.264} C_VEL
LIN {X 0,Y 276.479,Z 358.861,A -85,B 0,C 180,E1 -17537.147,E2 -17537.147} C_VEL
LIN {X 0,Y 277.245,Z 358.761,A -85,B 0,C 180,E1 -17541.337,E2 -17541.337} C_VEL
LIN {X 0,Y 277.511,Z 358.732,A -85,B 0,C 180,E1 -17544.184,E2 -17544.184} C_VEL
LIN {X 0,Y 277.813,Z 358.692,A -85,B 0,C 180,E1 -17548.549,E2 -17548.549} C_VEL
LIN {X 0,Y 277.812,Z 358.691,A -85,B 0,C 180,E1 -17551.448,E2 -17551.448} C_VEL
LIN {X 0,Y 277.644,Z 358.711,A -85,B 0,C 180,E1 -17557.269,E2 -17557.269} C_VEL
LIN {X 0,Y 277.496,Z 358.73,A -85,B 0,C 180,E1 -17560.21,E2 -17560.21} C_VEL
LIN {X 0,Y 277.424,Z 358.738,A -85,B 0,C 180,E1 -17564.673,E2 -17564.673} C_VEL
LIN {X 0,Y 277.333,Z 358.75,A -85,B 0,C 180,E1 -17569.233,E2 -17569.233} C_VEL
LIN {X 0,Y 277.316,Z 358.753,A -85,B 0,C 180,E1 -17573.919,E2 -17573.919} C_VEL
LIN {X 0,Y 277.313,Z 358.755,A -85,B 0,C 180,E1 -17577.504,E2 -17577.504} C_VEL
LIN {X 0,Y 277.259,Z 358.758,A -85,B 0,C 180,E1 -17580.481,E2 -17580.481} C_VEL
LIN {X 0,Y 277.241,Z 358.761,A -85,B 0,C 180,E1 -17583.894,E2 -17583.894} C_VEL
LIN {X 0,Y 277.279,Z 358.758,A -85,B 0,C 180,E1 -17587.465,E2 -17587.465} C_VEL
LIN {X 0,Y 277.281,Z 358.76,A -85,B 0,C 180,E1 -17591.221,E2 -17591.221} C_VEL
LIN {X 0,Y 277.274,Z 358.759,A -85,B 0,C 180,E1 -17595.208,E2 -17595.208} C_VEL
LIN {X 0,Y 277.282,Z 358.756,A -85,B 0,C 180,E1 -17599.494,E2 -17599.494} C_VEL
LIN {X 0,Y 277.278,Z 358.758,A -85,B 0,C 180,E1 -17602.535,E2 -17602.535} C_VEL
LIN {X 0,Y 277.24,Z 358.761,A -85,B 0,C 180,E1 -17606.106,E2 -17606.106} C_VEL
LIN {X 0,Y 277.248,Z 358.759,A -85,B 0,C 180,E1 -17609.539,E2 -17609.539} C_VEL
LIN {X 0,Y 277.346,Z 358.75,A -85,B 0,C 180,E1 -17612.865,E2 -17612.865} C_VEL
LIN {X 0,Y 277.367,Z 358.746,A -85,B 0,C 180,E1 -17616.085,E2 -17616.085} C_VEL
LIN {X 0,Y 277.364,Z 358.747,A -85,B 0,C 180,E1 -17620.769,E2 -17620.769} C_VEL
LIN {X 0,Y 277.423,Z 358.738,A -85,B 0,C 180,E1 -17625.327,E2 -17625.327} C_VEL
LIN {X 0,Y 277.495,Z 358.73,A -85,B 0,C 180,E1 -17629.79,E2 -17629.79} C_VEL
LIN {X 0,Y 277.642,Z 358.711,A -85,B 0,C 180,E1 -17632.73,E2 -17632.73} C_VEL
LIN {X 0,Y 277.811,Z 358.69,A -85,B 0,C 180,E1 -17638.552,E2 -17638.552} C_VEL
LIN {X 0,Y 277.813,Z 358.691,A -85,B 0,C 180,E1 -17641.451,E2 -17641.451} C_VEL
LIN {X 0,Y 277.643,Z 358.711,A -85,B 0,C 180,E1 -17647.273,E2 -17647.273} C_VEL
LIN {X 0,Y 277.498,Z 358.729,A -85,B 0,C 180,E1 -17650.213,E2 -17650.213} C_VEL
LIN {X 0,Y 277.426,Z 358.737,A -85,B 0,C 180,E1 -17654.676,E2 -17654.676} C_VEL
LIN {X 0,Y 277.425,Z 358.741,A -85,B 0,C 180,E1 -17655.826,E2 -17655.826} C_VEL
LIN {X 0,Y 276.669,Z 358.835,A -85,B 0,C 180,E1 -17657.038,E2 -17657.038} C_VEL
LIN {X 0,Y 273.732,Z 359.199,A -85,B 0,C 180,E1 -17659.01,E2 -17659.01} C_VEL
LIN {X 0,Y 271.295,Z 359.501,A -85,B 0,C 180,E1 -17660.613,E2 -17660.613} C_VEL
LIN {X 0,Y 270.27,Z 359.63,A -85,B 0,C 180,E1 -17661.857,E2 -17661.857} C_VEL
LIN {X 0,Y 270.195,Z 359.637,A -85,B 0,C 180,E1 -17662.278,E2 -17662.278} C_VEL
LIN {X 0,Y 270.267,Z 359.63,A -85,B 0,C 180,E1 -17664.588,E2 -17664.588} C_VEL
LIN {X 0,Y 270.265,Z 359.629,A -85,B 0,C 180,E1 -17667.911,E2 -17667.911} C_VEL
LIN {X 0,Y 270.178,Z 359.644,A -85,B 0,C 180,E1 -17671.35,E2 -17671.35} C_VEL
LIN {X 0,Y 270.195,Z 359.641,A -85,B 0,C 180,E1 -17674.908,E2 -17674.908} C_VEL
LIN {X 0,Y 270.192,Z 359.64,A -85,B 0,C 180,E1 -17678.713,E2 -17678.713} C_VEL
LIN {X 0,Y 270.167,Z 359.643,A -85,B 0,C 180,E1 -17683.253,E2 -17683.253} C_VEL
LIN {X 0,Y 270.248,Z 359.68,A -85,B 0,C 180,E1 -17688.043,E2 -17688.043} C_VEL
LIN {X 0,Y 271.297,Z 365.085,A -85,B 0,C 180,E1 -17692.503,E2 -17692.503} C_VEL
LIN {X 0,Y 271.85,Z 369.343,A -85,B 0,C 180,E1 -17695.822,E2 -17695.822} C_VEL
LIN {X 0,Y 271.325,Z 373.308,A -85,B 0,C 180,E1 -17698.737,E2 -17698.737} C_VEL
LIN {X 0,Y 270.264,Z 379.2,A -85,B 0,C 180,E1 -17702.933,E2 -17702.933} C_VEL
LIN {X 0,Y 269.388,Z 386.118,A -85,B 0,C 180,E1 -17707.775,E2 -17707.775} C_VEL
LIN {X 0,Y 268.997,Z 390.185,A -85,B 0,C 180,E1 -17710.456,E2 -17710.456} C_VEL
LIN {X 0,Y 270.472,Z 403.16,A -85,B 0,C 180,E1 -17711.343,E2 -17711.343} C_VEL
LIN {X 0,Y 271.319,Z 413.099,A -85,B 0,C 180,E1 -17712.284,E2 -17712.284} C_VEL
LIN {X 0,Y 271.879,Z 422.052,A -85,B 0,C 180,E1 -17713.348,E2 -17713.348} C_VEL
LIN {X 0,Y 272.057,Z 429.742,A -85,B 0,C 180,E1 -17714.456,E2 -17714.456} C_VEL
LIN {X 0,Y 270.993,Z 438.36,A -85,B 0,C 180,E1 -17715.931,E2 -17715.931} C_VEL
LIN {X 0,Y 270.095,Z 446.139,A -85,B 0,C 180,E1 -17717.606,E2 -17717.606} C_VEL
LIN {X 0,Y 269.299,Z 452.944,A -85,B 0,C 180,E1 -17719.476,E2 -17719.476} C_VEL
LIN {X 0,Y 268.871,Z 457.43,A -85,B 0,C 180,E1 -17720.979,E2 -17720.979} C_VEL
LIN {X 0,Y 268.541,Z 461.157,A -85,B 0,C 180,E1 -17722.483,E2 -17722.483} C_VEL
LIN {X 0,Y 268.289,Z 465.054,A -85,B 0,C 180,E1 -17724.53,E2 -17724.53} C_VEL
LIN {X 0,Y 268.289,Z 466.529,A -85,B 0,C 180,E1 -17725.495,E2 -17725.495} C_VEL
LIN {X 0,Y 268.33,Z 468.308,A -85,B 0,C 180,E1 -17726.999,E2 -17726.999} C_VEL
LIN {X 0,Y 268.293,Z 469.563,A -85,B 0,C 180,E1 -17728.501,E2 -17728.501} C_VEL
LIN {X 0,Y 268.328,Z 470.332,A -85,B 0,C 180,E1 -17730.002,E2 -17730.002} C_VEL
LIN {X 0,Y 268.277,Z 470.58,A -85,B 0,C 180,E1 -17731.503,E2 -17731.503} C_VEL
LIN {X 0,Y 268.275,Z 470.233,A -85,B 0,C 180,E1 -17733.005,E2 -17733.005} C_VEL
LIN {X 0,Y 268.249,Z 468.786,A -85,B 0,C 180,E1 -17735.38,E2 -17735.38} C_VEL
LIN {X 0,Y 268.549,Z 466.318,A -85,B 0,C 180,E1 -17737.521,E2 -17737.521} C_VEL
LIN {X 0,Y 269.18,Z 462.451,A -85,B 0,C 180,E1 -17739.773,E2 -17739.773} C_VEL
LIN {X 0,Y 270.152,Z 457.229,A -85,B 0,C 180,E1 -17742.014,E2 -17742.014} C_VEL
LIN {X 0,Y 271.32,Z 451.677,A -85,B 0,C 180,E1 -17743.865,E2 -17743.865} C_VEL
LIN {X 0,Y 272.808,Z 444.789,A -85,B 0,C 180,E1 -17745.696,E2 -17745.696} C_VEL
LIN {X 0,Y 274.486,Z 435.964,A -85,B 0,C 180,E1 -17747.51,E2 -17747.51} C_VEL
LIN {X 0,Y 275.091,Z 429.201,A -85,B 0,C 180,E1 -17748.695,E2 -17748.695} C_VEL
LIN {X 0,Y 275.126,Z 420.729,A -85,B 0,C 180,E1 -17749.98,E2 -17749.98} C_VEL
LIN {X 0,Y 274.647,Z 413.034,A -85,B 0,C 180,E1 -17750.995,E2 -17750.995} C_VEL
LIN {X 0,Y 273.445,Z 404.216,A -85,B 0,C 180,E1 -17752.022,E2 -17752.022} C_VEL
LIN {X 0,Y 271.539,Z 394.761,A -85,B 0,C 180,E1 -17752.989,E2 -17752.989} C_VEL
LIN {X 0,Y 269.867,Z 388.044,A -85,B 0,C 180,E1 -17753.621,E2 -17753.621} C_VEL
LIN {X 0,Y 270.909,Z 381.915,A -85,B 0,C 180,E1 -17758.109,E2 -17758.109} C_VEL
LIN {X 0,Y 272.292,Z 375.799,A -85,B 0,C 180,E1 -17762.823,E2 -17762.823} C_VEL
LIN {X 0,Y 272.439,Z 373.681,A -85,B 0,C 180,E1 -17764.58,E2 -17764.58} C_VEL
LIN {X 0,Y 272.191,Z 371.161,A -85,B 0,C 180,E1 -17766.828,E2 -17766.828} C_VEL
LIN {X 0,Y 271.595,Z 367.539,A -85,B 0,C 180,E1 -17770.312,E2 -17770.312} C_VEL
LIN {X 0,Y 270.868,Z 363.651,A -85,B 0,C 180,E1 -17774.473,E2 -17774.473} C_VEL
LIN {X 0,Y 270.474,Z 361.101,A -85,B 0,C 180,E1 -17777.499,E2 -17777.499} C_VEL
LIN {X 0,Y 270.186,Z 359.644,A -85,B 0,C 180,E1 -17779.435,E2 -17779.435} C_VEL
LIN {X 0,Y 270.235,Z 359.637,A -85,B 0,C 180,E1 -17783.731,E2 -17783.731} C_VEL
LIN {X 0,Y 270.211,Z 359.639,A -85,B 0,C 180,E1 -17786.892,E2 -17786.892} C_VEL
LIN {X 0,Y 270.204,Z 359.641,A -85,B 0,C 180,E1 -17790.382,E2 -17790.382} C_VEL
LIN {X 0,Y 270.271,Z 359.632,A -85,B 0,C 180,E1 -17793.763,E2 -17793.763} C_VEL
LIN {X 0,Y 270.242,Z 359.635,A -85,B 0,C 180,E1 -17797.038,E2 -17797.038} C_VEL
LIN {X 0,Y 270.31,Z 359.627,A -85,B 0,C 180,E1 -17800.244,E2 -17800.244} C_VEL
LIN {X 0,Y 270.412,Z 359.615,A -85,B 0,C 180,E1 -17804.935,E2 -17804.935} C_VEL
LIN {X 0,Y 270.418,Z 359.614,A -85,B 0,C 180,E1 -17809.517,E2 -17809.517} C_VEL
LIN {X 0,Y 270.578,Z 359.594,A -85,B 0,C 180,E1 -17812.537,E2 -17812.537} C_VEL
LIN {X 0,Y 270.792,Z 359.563,A -85,B 0,C 180,E1 -17818.511,E2 -17818.511} C_VEL
LIN {X 0,Y 270.793,Z 359.565,A -85,B 0,C 180,E1 -17821.486,E2 -17821.486} C_VEL
LIN {X 0,Y 270.59,Z 359.592,A -85,B 0,C 180,E1 -17827.46,E2 -17827.46} C_VEL
LIN {X 0,Y 270.415,Z 359.614,A -85,B 0,C 180,E1 -17830.48,E2 -17830.48} C_VEL
LIN {X 0,Y 270.338,Z 359.629,A -85,B 0,C 180,E1 -17833.529,E2 -17833.529} C_VEL
LIN {X 0,Y 270.413,Z 361.438,A -85,B 0,C 180,E1 -17836.61,E2 -17836.61} C_VEL
LIN {X 0,Y 270.219,Z 364.093,A -85,B 0,C 180,E1 -17840.556,E2 -17840.556} C_VEL
LIN {X 0,Y 269.823,Z 367.08,A -85,B 0,C 180,E1 -17844.627,E2 -17844.627} C_VEL
LIN {X 0,Y 269.677,Z 368.603,A -85,B 0,C 180,E1 -17846.508,E2 -17846.508} C_VEL
LIN {X 0,Y 271.662,Z 374.366,A -85,B 0,C 180,E1 -17847.143,E2 -17847.143} C_VEL
LIN {X 0,Y 274.935,Z 385.175,A -85,B 0,C 180,E1 -17848.454,E2 -17848.454} C_VEL
LIN {X 0,Y 277.001,Z 395.008,A -85,B 0,C 180,E1 -17849.831,E2 -17849.831} C_VEL
LIN {X 0,Y 277.825,Z 402.292,A -85,B 0,C 180,E1 -17850.96,E2 -17850.96} C_VEL
LIN {X 0,Y 276.506,Z 410.457,A -85,B 0,C 180,E1 -17852.258,E2 -17852.258} C_VEL
LIN {X 0,Y 275.256,Z 416.805,A -85,B 0,C 180,E1 -17853.468,E2 -17853.468} C_VEL
LIN {X 0,Y 274.083,Z 422.819,A -85,B 0,C 180,E1 -17854.859,E2 -17854.859} C_VEL
LIN {X 0,Y 272.9,Z 428.091,A -85,B 0,C 180,E1 -17856.319,E2 -17856.319} C_VEL
LIN {X 0,Y 271.911,Z 432.295,A -85,B 0,C 180,E1 -17857.707,E2 -17857.707} C_VEL
LIN {X 0,Y 270.71,Z 437.259,A -85,B 0,C 180,E1 -17859.812,E2 -17859.812} C_VEL
LIN {X 0,Y 270.108,Z 439.597,A -85,B 0,C 180,E1 -17861.011,E2 -17861.011} C_VEL
LIN {X 0,Y 269.326,Z 442.538,A -85,B 0,C 180,E1 -17863.057,E2 -17863.057} C_VEL
LIN {X 0,Y 268.746,Z 444.455,A -85,B 0,C 180,E1 -17865.081,E2 -17865.081} C_VEL
LIN {X 0,Y 268.33,Z 445.456,A -85,B 0,C 180,E1 -17867.166,E2 -17867.166} C_VEL
LIN {X 0,Y 268.086,Z 445.44,A -85,B 0,C 180,E1 -17869.483,E2 -17869.483} C_VEL
LIN {X 0,Y 268.141,Z 444.238,A -85,B 0,C 180,E1 -17871.838,E2 -17871.838} C_VEL
LIN {X 0,Y 268.452,Z 441.721,A -85,B 0,C 180,E1 -17874.246,E2 -17874.246} C_VEL
LIN {X 0,Y 268.689,Z 439.326,A -85,B 0,C 180,E1 -17875.778,E2 -17875.778} C_VEL
LIN {X 0,Y 269.298,Z 434.467,A -85,B 0,C 180,E1 -17878.104,E2 -17878.104} C_VEL
LIN {X 0,Y 269.858,Z 429.731,A -85,B 0,C 180,E1 -17879.842,E2 -17879.842} C_VEL
LIN {X 0,Y 270.663,Z 423.663,A -85,B 0,C 180,E1 -17881.624,E2 -17881.624} C_VEL
LIN {X 0,Y 271.475,Z 416.758,A -85,B 0,C 180,E1 -17883.267,E2 -17883.267} C_VEL
LIN {X 0,Y 272.335,Z 410.017,A -85,B 0,C 180,E1 -17884.58,E2 -17884.58} C_VEL
LIN {X 0,Y 273.241,Z 401.808,A -85,B 0,C 180,E1 -17885.899,E2 -17885.899} C_VEL
LIN {X 0,Y 273.826,Z 395.304,A -85,B 0,C 180,E1 -17886.756,E2 -17886.756} C_VEL
LIN {X 0,Y 272.823,Z 387.796,A -85,B 0,C 180,E1 -17887.667,E2 -17887.667} C_VEL
LIN {X 0,Y 271.018,Z 377.344,A -85,B 0,C 180,E1 -17888.711,E2 -17888.711} C_VEL
LIN {X 0,Y 268.832,Z 366.477,A -85,B 0,C 180,E1 -17889.564,E2 -17889.564} C_VEL
LIN {X 0,Y 269.03,Z 363.071,A -85,B 0,C 180,E1 -17893.298,E2 -17893.298} C_VEL
LIN {X 0,Y 269.423,Z 359.74,A -85,B 0,C 180,E1 -17897.188,E2 -17897.188} C_VEL
LIN {X 0,Y 270.2,Z 359.638,A -85,B 0,C 180,E1 -17901.248,E2 -17901.248} C_VEL
LIN {X 0,Y 270.473,Z 359.608,A -85,B 0,C 180,E1 -17904.032,E2 -17904.032} C_VEL
LIN {X 0,Y 270.779,Z 359.568,A -85,B 0,C 180,E1 -17908.511,E2 -17908.511} C_VEL
LIN {X 0,Y 270.778,Z 359.567,A -85,B 0,C 180,E1 -17911.485,E2 -17911.485} C_VEL
LIN {X 0,Y 270.602,Z 359.589,A -85,B 0,C 180,E1 -17917.459,E2 -17917.459} C_VEL
LIN {X 0,Y 270.431,Z 359.608,A -85,B 0,C 180,E1 -17920.479,E2 -17920.479} C_VEL
LIN {X 0,Y 270.392,Z 359.614,A -85,B 0,C 180,E1 -17925.063,E2 -17925.063} C_VEL
LIN {X 0,Y 270.29,Z 359.629,A -85,B 0,C 180,E1 -17929.754,E2 -17929.754} C_VEL
LIN {X 0,Y 270.262,Z 359.63,A -85,B 0,C 180,E1 -17934.584,E2 -17934.584} C_VEL
LIN {X 0,Y 270.258,Z 359.63,A -85,B 0,C 180,E1 -17937.908,E2 -17937.908} C_VEL
LIN {X 0,Y 270.171,Z 359.646,A -85,B 0,C 180,E1 -17941.347,E2 -17941.347} C_VEL
LIN {X 0,Y 270.203,Z 359.639,A -85,B 0,C 180,E1 -17944.903,E2 -17944.903} C_VEL
LIN {X 0,Y 270.239,Z 359.634,A -85,B 0,C 180,E1 -17948.725,E2 -17948.725} C_VEL
LIN {X 0,Y 270.243,Z 359.633,A -85,B 0,C 180,E1 -17952.541,E2 -17952.541} C_VEL
LIN {X 0,Y 270.219,Z 359.637,A -85,B 0,C 180,E1 -17956.736,E2 -17956.736} C_VEL
LIN {X 0,Y 270.236,Z 359.634,A -85,B 0,C 180,E1 -17959.448,E2 -17959.448} C_VEL
LIN {X 0,Y 270.244,Z 359.631,A -85,B 0,C 180,E1 -17963.721,E2 -17963.721} C_VEL
LIN {X 0,Y 270.19,Z 359.643,A -85,B 0,C 180,E1 -17966.893,E2 -17966.893} C_VEL
LIN {X 0,Y 270.215,Z 359.638,A -85,B 0,C 180,E1 -17970.387,E2 -17970.387} C_VEL
LIN {X 0,Y 270.256,Z 359.631,A -85,B 0,C 180,E1 -17973.765,E2 -17973.765} C_VEL
LIN {X 0,Y 270.264,Z 359.63,A -85,B 0,C 180,E1 -17977.044,E2 -17977.044} C_VEL
LIN {X 0,Y 270.319,Z 359.624,A -85,B 0,C 180,E1 -17980.248,E2 -17980.248} C_VEL
LIN {X 0,Y 270.391,Z 359.614,A -85,B 0,C 180,E1 -17984.936,E2 -17984.936} C_VEL
LIN {X 0,Y 270.43,Z 359.609,A -85,B 0,C 180,E1 -17989.52,E2 -17989.52} C_VEL
LIN {X 0,Y 270.6,Z 359.59,A -85,B 0,C 180,E1 -17992.54,E2 -17992.54} C_VEL
LIN {X 0,Y 270.777,Z 359.567,A -85,B 0,C 180,E1 -17998.514,E2 -17998.514} C_VEL
LIN {X 0,Y 270.779,Z 359.567,A -85,B 0,C 180,E1 -18001.489,E2 -18001.489} C_VEL
LIN {X 0,Y 270.602,Z 359.59,A -85,B 0,C 180,E1 -18007.463,E2 -18007.463} C_VEL
LIN {X 0,Y 270.433,Z 359.608,A -85,B 0,C 180,E1 -18010.483,E2 -18010.483} C_VEL
LIN {X 0,Y 270.395,Z 359.614,A -85,B 0,C 180,E1 -18015.066,E2 -18015.066} C_VEL
LIN {X 0,Y 270.293,Z 359.627,A -85,B 0,C 180,E1 -18019.757,E2 -18019.757} C_VEL
LIN {X 0,Y 270.195,Z 359.637,A -85,B 0,C 180,E1 -18022.278,E2 -18022.278} C_VEL
LIN {X 0,Y 269.562,Z 359.721,A -85,B 0,C 180,E1 -18023.522,E2 -18023.522} C_VEL
LIN {X 0,Y 266.765,Z 360.072,A -85,B 0,C 180,E1 -18025.549,E2 -18025.549} C_VEL
LIN {X 0,Y 264.347,Z 360.373,A -85,B 0,C 180,E1 -18027.197,E2 -18027.197} C_VEL
LIN {X 0,Y 263.268,Z 360.503,A -85,B 0,C 180,E1 -18028.474,E2 -18028.474} C_VEL
LIN {X 0,Y 263.159,Z 360.513,A -85,B 0,C 180,E1 -18028.907,E2 -18028.907} C_VEL
LIN {X 0,Y 263.127,Z 360.519,A -85,B 0,C 180,E1 -18032.29,E2 -18032.29} C_VEL
LIN {X 0,Y 263.176,Z 360.514,A -85,B 0,C 180,E1 -18036.765,E2 -18036.765} C_VEL
LIN {X 0,Y 263.12,Z 360.52,A -85,B 0,C 180,E1 -18041.596,E2 -18041.596} C_VEL
LIN {X 0,Y 263.13,Z 360.518,A -85,B 0,C 180,E1 -18046.021,E2 -18046.021} C_VEL
LIN {X 0,Y 263.23,Z 360.575,A -85,B 0,C 180,E1 -18047.873,E2 -18047.873} C_VEL
LIN {X 0,Y 264.227,Z 365.785,A -85,B 0,C 180,E1 -18052.286,E2 -18052.286} C_VEL
LIN {X 0,Y 264.805,Z 369.602,A -85,B 0,C 180,E1 -18055.363,E2 -18055.363} C_VEL
LIN {X 0,Y 264.456,Z 372.917,A -85,B 0,C 180,E1 -18057.895,E2 -18057.895} C_VEL
LIN {X 0,Y 263.508,Z 378.039,A -85,B 0,C 180,E1 -18061.661,E2 -18061.661} C_VEL
LIN {X 0,Y 262.496,Z 384.458,A -85,B 0,C 180,E1 -18066.324,E2 -18066.324} C_VEL
LIN {X 0,Y 261.947,Z 389.641,A -85,B 0,C 180,E1 -18070.023,E2 -18070.023} C_VEL
LIN {X 0,Y 263.442,Z 402.835,A -85,B 0,C 180,E1 -18070.969,E2 -18070.969} C_VEL
LIN {X 0,Y 264.141,Z 411.412,A -85,B 0,C 180,E1 -18071.785,E2 -18071.785} C_VEL
LIN {X 0,Y 264.788,Z 420.345,A -85,B 0,C 180,E1 -18072.848,E2 -18072.848} C_VEL
LIN {X 0,Y 265.056,Z 428.549,A -85,B 0,C 180,E1 -18074.035,E2 -18074.035} C_VEL
LIN {X 0,Y 264.444,Z 435.312,A -85,B 0,C 180,E1 -18075.181,E2 -18075.181} C_VEL
LIN {X 0,Y 263.535,Z 441.892,A -85,B 0,C 180,E1 -18076.508,E2 -18076.508} C_VEL
LIN {X 0,Y 262.778,Z 448.17,A -85,B 0,C 180,E1 -18078.039,E2 -18078.039} C_VEL
LIN {X 0,Y 262.155,Z 453.383,A -85,B 0,C 180,E1 -18079.577,E2 -18079.577} C_VEL
LIN {X 0,Y 261.828,Z 456.766,A -85,B 0,C 180,E1 -18080.734,E2 -18080.734} C_VEL
LIN {X 0,Y 261.503,Z 460.551,A -85,B 0,C 180,E1 -18082.279,E2 -18082.279} C_VEL
LIN {X 0,Y 261.199,Z 464.845,A -85,B 0,C 180,E1 -18084.599,E2 -18084.599} C_VEL
LIN {X 0,Y 261.258,Z 467.835,A -85,B 0,C 180,E1 -18086.918,E2 -18086.918} C_VEL
LIN {X 0,Y 261.218,Z 469.146,A -85,B 0,C 180,E1 -18088.46,E2 -18088.46} C_VEL
LIN {X 0,Y 261.248,Z 469.968,A -85,B 0,C 180,E1 -18090.002,E2 -18090.002} C_VEL
LIN {X 0,Y 261.201,Z 470.227,A -85,B 0,C 180,E1 -18091.544,E2 -18091.544} C_VEL
LIN {X 0,Y 261.183,Z 469.921,A -85,B 0,C 180,E1 -18093.087,E2 -18093.087} C_VEL
LIN {X 0,Y 261.164,Z 468.681,A -85,B 0,C 180,E1 -18095.317,E2 -18095.317} C_VEL
LIN {X 0,Y 261.494,Z 466.162,A -85,B 0,C 180,E1 -18097.725,E2 -18097.725} C_VEL
LIN {X 0,Y 262.157,Z 462.386,A -85,B 0,C 180,E1 -18100.037,E2 -18100.037} C_VEL
LIN {X 0,Y 262.803,Z 459.19,A -85,B 0,C 180,E1 -18101.572,E2 -18101.572} C_VEL
LIN {X 0,Y 263.911,Z 454.142,A -85,B 0,C 180,E1 -18103.476,E2 -18103.476} C_VEL
LIN {X 0,Y 265.278,Z 447.846,A -85,B 0,C 180,E1 -18105.365,E2 -18105.365} C_VEL
LIN {X 0,Y 266.646,Z 441.731,A -85,B 0,C 180,E1 -18106.855,E2 -18106.855} C_VEL
LIN {X 0,Y 267.872,Z 435.37,A -85,B 0,C 180,E1 -18108.155,E2 -18108.155} C_VEL
LIN {X 0,Y 268.412,Z 428.916,A -85,B 0,C 180,E1 -18109.32,E2 -18109.32} C_VEL
LIN {X 0,Y 268.412,Z 420.106,A -85,B 0,C 180,E1 -18110.702,E2 -18110.702} C_VEL
LIN {X 0,Y 267.904,Z 412.801,A -85,B 0,C 180,E1 -18111.712,E2 -18111.712} C_VEL
LIN {X 0,Y 266.761,Z 404.18,A -85,B 0,C 180,E1 -18112.763,E2 -18112.763} C_VEL
LIN {X 0,Y 264.645,Z 394.209,A -85,B 0,C 180,E1 -18113.838,E2 -18113.838} C_VEL
LIN {X 0,Y 263.025,Z 387.929,A -85,B 0,C 180,E1 -18114.441,E2 -18114.441} C_VEL
LIN {X 0,Y 263.045,Z 387.342,A -85,B 0,C 180,E1 -18114.712,E2 -18114.712} C_VEL
LIN {X 0,Y 264.235,Z 381.123,A -85,B 0,C 180,E1 -18119.478,E2 -18119.478} C_VEL
LIN {X 0,Y 265.267,Z 376.843,A -85,B 0,C 180,E1 -18122.899,E2 -18122.899} C_VEL
LIN {X 0,Y 265.366,Z 373.705,A -85,B 0,C 180,E1 -18125.639,E2 -18125.639} C_VEL
LIN {X 0,Y 264.731,Z 369.552,A -85,B 0,C 180,E1 -18129.655,E2 -18129.655} C_VEL
LIN {X 0,Y 264.36,Z 367.432,A -85,B 0,C 180,E1 -18131.893,E2 -18131.893} C_VEL
LIN {X 0,Y 263.69,Z 363.732,A -85,B 0,C 180,E1 -18136.133,E2 -18136.133} C_VEL
LIN {X 0,Y 263.134,Z 360.522,A -85,B 0,C 180,E1 -18140.466,E2 -18140.466} C_VEL
LIN {X 0,Y 263.172,Z 360.517,A -85,B 0,C 180,E1 -18144.018,E2 -18144.018} C_VEL
LIN {X 0,Y 263.141,Z 360.521,A -85,B 0,C 180,E1 -18147.712,E2 -18147.712} C_VEL
LIN {X 0,Y 263.205,Z 360.514,A -85,B 0,C 180,E1 -18151.785,E2 -18151.785} C_VEL
LIN {X 0,Y 263.235,Z 360.508,A -85,B 0,C 180,E1 -18155.2,E2 -18155.2} C_VEL
LIN {X 0,Y 263.273,Z 360.503,A -85,B 0,C 180,E1 -18159.693,E2 -18159.693} C_VEL
LIN {X 0,Y 263.36,Z 360.492,A -85,B 0,C 180,E1 -18164.521,E2 -18164.521} C_VEL
LIN {X 0,Y 263.358,Z 360.493,A -85,B 0,C 180,E1 -18169.232,E2 -18169.232} C_VEL
LIN {X 0,Y 263.54,Z 360.47,A -85,B 0,C 180,E1 -18172.336,E2 -18172.336} C_VEL
LIN {X 0,Y 263.756,Z 360.44,A -85,B 0,C 180,E1 -18178.472,E2 -18178.472} C_VEL
LIN {X 0,Y 263.757,Z 360.441,A -85,B 0,C 180,E1 -18181.525,E2 -18181.525} C_VEL
LIN {X 0,Y 263.55,Z 360.469,A -85,B 0,C 180,E1 -18187.661,E2 -18187.661} C_VEL
LIN {X 0,Y 263.354,Z 360.494,A -85,B 0,C 180,E1 -18190.765,E2 -18190.765} C_VEL
LIN {X 0,Y 263.319,Z 360.5,A -85,B 0,C 180,E1 -18192.327,E2 -18192.327} C_VEL
LIN {X 0,Y 263.362,Z 361.023,A -85,B 0,C 180,E1 -18193.895,E2 -18193.895} C_VEL
LIN {X 0,Y 263.383,Z 362.972,A -85,B 0,C 180,E1 -18197.067,E2 -18197.067} C_VEL
LIN {X 0,Y 263.174,Z 365.448,A -85,B 0,C 180,E1 -18200.822,E2 -18200.822} C_VEL
LIN {X 0,Y 262.708,Z 368.703,A -85,B 0,C 180,E1 -18205.341,E2 -18205.341} C_VEL
LIN {X 0,Y 262.711,Z 368.892,A -85,B 0,C 180,E1 -18205.606,E2 -18205.606} C_VEL
LIN {X 0,Y 263.745,Z 372.011,A -85,B 0,C 180,E1 -18205.975,E2 -18205.975} C_VEL
LIN {X 0,Y 266.446,Z 379.738,A -85,B 0,C 180,E1 -18206.926,E2 -18206.926} C_VEL
LIN {X 0,Y 269.072,Z 389.477,A -85,B 0,C 180,E1 -18208.254,E2 -18208.254} C_VEL
LIN {X 0,Y 270.479,Z 396.849,A -85,B 0,C 180,E1 -18209.367,E2 -18209.367} C_VEL
LIN {X 0,Y 271.212,Z 403.98,A -85,B 0,C 180,E1 -18210.549,E2 -18210.549} C_VEL
LIN {X 0,Y 269.758,Z 411.94,A -85,B 0,C 180,E1 -18211.877,E2 -18211.877} C_VEL
LIN {X 0,Y 268.473,Z 418.04,A -85,B 0,C 180,E1 -18213.101,E2 -18213.101} C_VEL
LIN {X 0,Y 267.05,Z 424.713,A -85,B 0,C 180,E1 -18214.741,E2 -18214.741} C_VEL
LIN {X 0,Y 265.719,Z 430.161,A -85,B 0,C 180,E1 -18216.383,E2 -18216.383} C_VEL
LIN {X 0,Y 264.372,Z 435.778,A -85,B 0,C 180,E1 -18218.519,E2 -18218.519} C_VEL
LIN {X 0,Y 263.188,Z 439.975,A -85,B 0,C 180,E1 -18220.643,E2 -18220.643} C_VEL
LIN {X 0,Y 262.637,Z 441.936,A -85,B 0,C 180,E1 -18221.986,E2 -18221.986} C_VEL
LIN {X 0,Y 261.895,Z 444.408,A -85,B 0,C 180,E1 -18224.241,E2 -18224.241} C_VEL
LIN {X 0,Y 261.342,Z 445.734,A -85,B 0,C 180,E1 -18226.556,E2 -18226.556} C_VEL
LIN {X 0,Y 261.025,Z 445.884,A -85,B 0,C 180,E1 -18228.925,E2 -18228.925} C_VEL
LIN {X 0,Y 261.042,Z 444.591,A -85,B 0,C 180,E1 -18231.738,E2 -18231.738} C_VEL
LIN {X 0,Y 261.272,Z 442.57,A -85,B 0,C 180,E1 -18233.798,E2 -18233.798} C_VEL
LIN {X 0,Y 261.714,Z 438.688,A -85,B 0,C 180,E1 -18236.349,E2 -18236.349} C_VEL
LIN {X 0,Y 262.269,Z 434.47,A -85,B 0,C 180,E1 -18238.325,E2 -18238.325} C_VEL
LIN {X 0,Y 262.78,Z 430.299,A -85,B 0,C 180,E1 -18239.901,E2 -18239.901} C_VEL
LIN {X 0,Y 263.553,Z 424.629,A -85,B 0,C 180,E1 -18241.637,E2 -18241.637} C_VEL
LIN {X 0,Y 264.28,Z 418.758,A -85,B 0,C 180,E1 -18243.121,E2 -18243.121} C_VEL
LIN {X 0,Y 265.226,Z 411.403,A -85,B 0,C 180,E1 -18244.644,E2 -18244.644} C_VEL
LIN {X 0,Y 266.042,Z 404.502,A -85,B 0,C 180,E1 -18245.827,E2 -18245.827} C_VEL
LIN {X 0,Y 266.837,Z 396.705,A -85,B 0,C 180,E1 -18246.933,E2 -18246.933} C_VEL
LIN {X 0,Y 265.958,Z 389.311,A -85,B 0,C 180,E1 -18247.877,E2 -18247.877} C_VEL
LIN {X 0,Y 264.565,Z 380.924,A -85,B 0,C 180,E1 -18248.779,E2 -18248.779} C_VEL
LIN {X 0,Y 262.725,Z 371.462,A -85,B 0,C 180,E1 -18249.597,E2 -18249.597} C_VEL
LIN {X 0,Y 261.786,Z 366.779,A -85,B 0,C 180,E1 -18249.982,E2 -18249.982} C_VEL
LIN {X 0,Y 262.122,Z 362.448,A -85,B 0,C 180,E1 -18254.838,E2 -18254.838} C_VEL
LIN {X 0,Y 262.335,Z 360.623,A -85,B 0,C 180,E1 -18257.032,E2 -18257.032} C_VEL
LIN {X 0,Y 263.133,Z 360.519,A -85,B 0,C 180,E1 -18261.186,E2 -18261.186} C_VEL
LIN {X 0,Y 263.434,Z 360.484,A -85,B 0,C 180,E1 -18263.872,E2 -18263.872} C_VEL
LIN {X 0,Y 263.743,Z 360.445,A -85,B 0,C 180,E1 -18268.471,E2 -18268.471} C_VEL
LIN {X 0,Y 263.743,Z 360.444,A -85,B 0,C 180,E1 -18271.525,E2 -18271.525} C_VEL
LIN {X 0,Y 263.563,Z 360.467,A -85,B 0,C 180,E1 -18277.66,E2 -18277.66} C_VEL
LIN {X 0,Y 263.364,Z 360.488,A -85,B 0,C 180,E1 -18280.764,E2 -18280.764} C_VEL
LIN {X 0,Y 263.34,Z 360.495,A -85,B 0,C 180,E1 -18285.476,E2 -18285.476} C_VEL
LIN {X 0,Y 263.252,Z 360.502,A -85,B 0,C 180,E1 -18290.305,E2 -18290.305} C_VEL
LIN {X 0,Y 263.196,Z 360.513,A -85,B 0,C 180,E1 -18295.29,E2 -18295.29} C_VEL
LIN {X 0,Y 263.163,Z 360.513,A -85,B 0,C 180,E1 -18298.729,E2 -18298.729} C_VEL
LIN {X 0,Y 263.12,Z 360.52,A -85,B 0,C 180,E1 -18302.287,E2 -18302.287} C_VEL
LIN {X 0,Y 263.177,Z 360.511,A -85,B 0,C 180,E1 -18305.977,E2 -18305.977} C_VEL
LIN {X 0,Y 263.18,Z 360.513,A -85,B 0,C 180,E1 -18309.856,E2 -18309.856} C_VEL
LIN {X 0,Y 263.177,Z 360.511,A -85,B 0,C 180,E1 -18313.969,E2 -18313.969} C_VEL
LIN {X 0,Y 263.199,Z 360.511,A -85,B 0,C 180,E1 -18318.385,E2 -18318.385} C_VEL
LIN {X 0,Y 263.193,Z 360.511,A -85,B 0,C 180,E1 -18323.23,E2 -18323.23} C_VEL
LIN {X 0,Y 263.17,Z 360.513,A -85,B 0,C 180,E1 -18325.891,E2 -18325.891} C_VEL
LIN {X 0,Y 263.137,Z 360.517,A -85,B 0,C 180,E1 -18329.507,E2 -18329.507} C_VEL
LIN {X 0,Y 263.183,Z 360.513,A -85,B 0,C 180,E1 -18333.004,E2 -18333.004} C_VEL
LIN {X 0,Y 263.213,Z 360.512,A -85,B 0,C 180,E1 -18336.392,E2 -18336.392} C_VEL
LIN {X 0,Y 263.281,Z 360.498,A -85,B 0,C 180,E1 -18339.697,E2 -18339.697} C_VEL
LIN {X 0,Y 263.339,Z 360.495,A -85,B 0,C 180,E1 -18344.523,E2 -18344.523} C_VEL
LIN {X 0,Y 263.363,Z 360.489,A -85,B 0,C 180,E1 -18349.236,E2 -18349.236} C_VEL
LIN {X 0,Y 263.561,Z 360.468,A -85,B 0,C 180,E1 -18352.34,E2 -18352.34} C_VEL
LIN {X 0,Y 263.741,Z 360.444,A -85,B 0,C 180,E1 -18358.475,E2 -18358.475} C_VEL
LIN {X 0,Y 263.743,Z 360.444,A -85,B 0,C 180,E1 -18361.528,E2 -18361.528} C_VEL
LIN {X 0,Y 263.563,Z 360.468,A -85,B 0,C 180,E1 -18367.663,E2 -18367.663} C_VEL
LIN {X 0,Y 263.365,Z 360.489,A -85,B 0,C 180,E1 -18370.767,E2 -18370.767} C_VEL
LIN {X 0,Y 263.342,Z 360.495,A -85,B 0,C 180,E1 -18375.48,E2 -18375.48} C_VEL
LIN {X 0,Y 263.256,Z 360.501,A -85,B 0,C 180,E1 -18380.309,E2 -18380.309} C_VEL
LIN {X 0,Y 263.202,Z 360.514,A -85,B 0,C 180,E1 -18385.293,E2 -18385.293} C_VEL
LIN {X 0,Y 263.159,Z 360.513,A -85,B 0,C 180,E1 -18388.907,E2 -18388.907} C_VEL
LIN {X 0,Y 262.434,Z 360.605,A -85,B 0,C 180,E1 -18390.184,E2 -18390.184} C_VEL
LIN {X 0,Y 259.567,Z 360.962,A -85,B 0,C 180,E1 -18392.267,E2 -18392.267} C_VEL
LIN {X 0,Y 257.169,Z 361.264,A -85,B 0,C 180,E1 -18393.961,E2 -18393.961} C_VEL
LIN {X 0,Y 256.144,Z 361.391,A -85,B 0,C 180,E1 -18395.274,E2 -18395.274} C_VEL
LIN {X 0,Y 256.06,Z 361.398,A -85,B 0,C 180,E1 -18395.719,E2 -18395.719} C_VEL
LIN {X 0,Y 256.066,Z 361.402,A -85,B 0,C 180,E1 -18399.144,E2 -18399.144} C_VEL
LIN {X 0,Y 256.061,Z 361.4,A -85,B 0,C 180,E1 -18403.329,E2 -18403.329} C_VEL
LIN {X 0,Y 256.179,Z 361.575,A -85,B 0,C 180,E1 -18407.794,E2 -18407.794} C_VEL
LIN {X 0,Y 257.219,Z 366.868,A -85,B 0,C 180,E1 -18412.409,E2 -18412.409} C_VEL
LIN {X 0,Y 257.707,Z 370.066,A -85,B 0,C 180,E1 -18415.064,E2 -18415.064} C_VEL
LIN {X 0,Y 257.387,Z 373.584,A -85,B 0,C 180,E1 -18417.83,E2 -18417.83} C_VEL
LIN {X 0,Y 256.537,Z 378.083,A -85,B 0,C 180,E1 -18421.244,E2 -18421.244} C_VEL
LIN {X 0,Y 255.403,Z 385.108,A -85,B 0,C 180,E1 -18426.487,E2 -18426.487} C_VEL
LIN {X 0,Y 254.903,Z 389.373,A -85,B 0,C 180,E1 -18429.626,E2 -18429.626} C_VEL
LIN {X 0,Y 256.313,Z 401.614,A -85,B 0,C 180,E1 -18430.494,E2 -18430.494} C_VEL
LIN {X 0,Y 257.134,Z 411.629,A -85,B 0,C 180,E1 -18431.476,E2 -18431.476} C_VEL
LIN {X 0,Y 257.77,Z 420.728,A -85,B 0,C 180,E1 -18432.607,E2 -18432.607} C_VEL
LIN {X 0,Y 258.028,Z 428.728,A -85,B 0,C 180,E1 -18433.813,E2 -18433.813} C_VEL
LIN {X 0,Y 257.424,Z 435.296,A -85,B 0,C 180,E1 -18434.97,E2 -18434.97} C_VEL
LIN {X 0,Y 256.58,Z 440.969,A -85,B 0,C 180,E1 -18436.135,E2 -18436.135} C_VEL
LIN {X 0,Y 255.812,Z 447.348,A -85,B 0,C 180,E1 -18437.709,E2 -18437.709} C_VEL
LIN {X 0,Y 255.147,Z 452.644,A -85,B 0,C 180,E1 -18439.287,E2 -18439.287} C_VEL
LIN {X 0,Y 254.601,Z 458.021,A -85,B 0,C 180,E1 -18441.27,E2 -18441.27} C_VEL
LIN {X 0,Y 254.314,Z 461.489,A -85,B 0,C 180,E1 -18442.858,E2 -18442.858} C_VEL
LIN {X 0,Y 254.103,Z 465.462,A -85,B 0,C 180,E1 -18445.243,E2 -18445.243} C_VEL
LIN {X 0,Y 254.165,Z 467.359,A -85,B 0,C 180,E1 -18446.832,E2 -18446.832} C_VEL
LIN {X 0,Y 254.145,Z 468.726,A -85,B 0,C 180,E1 -18448.417,E2 -18448.417} C_VEL
LIN {X 0,Y 254.171,Z 469.594,A -85,B 0,C 180,E1 -18450.002,E2 -18450.002} C_VEL
LIN {X 0,Y 254.127,Z 469.861,A -85,B 0,C 180,E1 -18451.587,E2 -18451.587} C_VEL
LIN {X 0,Y 254.093,Z 469.611,A -85,B 0,C 180,E1 -18453.173,E2 -18453.173} C_VEL
LIN {X 0,Y 254.09,Z 468.556,A -85,B 0,C 180,E1 -18455.281,E2 -18455.281} C_VEL
LIN {X 0,Y 254.43,Z 466.005,A -85,B 0,C 180,E1 -18457.941,E2 -18457.941} C_VEL
LIN {X 0,Y 255.152,Z 462.333,A -85,B 0,C 180,E1 -18460.316,E2 -18460.316} C_VEL
LIN {X 0,Y 255.835,Z 459.188,A -85,B 0,C 180,E1 -18461.892,E2 -18461.892} C_VEL
LIN {X 0,Y 257.236,Z 453.057,A -85,B 0,C 180,E1 -18464.236,E2 -18464.236} C_VEL
LIN {X 0,Y 258.45,Z 448.032,A -85,B 0,C 180,E1 -18465.781,E2 -18465.781} C_VEL
LIN {X 0,Y 259.88,Z 442.042,A -85,B 0,C 180,E1 -18467.308,E2 -18467.308} C_VEL
LIN {X 0,Y 261.28,Z 434.836,A -85,B 0,C 180,E1 -18468.833,E2 -18468.833} C_VEL
LIN {X 0,Y 261.772,Z 427.386,A -85,B 0,C 180,E1 -18470.211,E2 -18470.211} C_VEL
LIN {X 0,Y 261.74,Z 419.615,A -85,B 0,C 180,E1 -18471.462,E2 -18471.462} C_VEL
LIN {X 0,Y 261.057,Z 411.279,A -85,B 0,C 180,E1 -18472.646,E2 -18472.646} C_VEL
LIN {X 0,Y 260.021,Z 403.731,A -85,B 0,C 180,E1 -18473.595,E2 -18473.595} C_VEL
LIN {X 0,Y 257.764,Z 393.659,A -85,B 0,C 180,E1 -18474.754,E2 -18474.754} C_VEL
LIN {X 0,Y 256.149,Z 387.195,A -85,B 0,C 180,E1 -18475.464,E2 -18475.464} C_VEL
LIN {X 0,Y 257.431,Z 381.085,A -85,B 0,C 180,E1 -18480.337,E2 -18480.337} C_VEL
LIN {X 0,Y 258.246,Z 377.886,A -85,B 0,C 180,E1 -18482.978,E2 -18482.978} C_VEL
LIN {X 0,Y 258.391,Z 375.278,A -85,B 0,C 180,E1 -18485.315,E2 -18485.315} C_VEL
LIN {X 0,Y 257.939,Z 371.711,A -85,B 0,C 180,E1 -18488.807,E2 -18488.807} C_VEL
LIN {X 0,Y 257.174,Z 367.78,A -85,B 0,C 180,E1 -18493.096,E2 -18493.096} C_VEL
LIN {X 0,Y 256.64,Z 364.752,A -85,B 0,C 180,E1 -18496.793,E2 -18496.793} C_VEL
LIN {X 0,Y 256.152,Z 361.823,A -85,B 0,C 180,E1 -18500.871,E2 -18500.871} C_VEL
LIN {X 0,Y 256.12,Z 361.395,A -85,B 0,C 180,E1 -18501.869,E2 -18501.869} C_VEL
LIN {X 0,Y 256.114,Z 361.396,A -85,B 0,C 180,E1 -18505.412,E2 -18505.412} C_VEL
LIN {X 0,Y 256.101,Z 361.397,A -85,B 0,C 180,E1 -18508.572,E2 -18508.572} C_VEL
LIN {X 0,Y 256.147,Z 361.391,A -85,B 0,C 180,E1 -18512.195,E2 -18512.195} C_VEL
LIN {X 0,Y 256.176,Z 361.388,A -85,B 0,C 180,E1 -18515.699,E2 -18515.699} C_VEL
LIN {X 0,Y 256.176,Z 361.389,A -85,B 0,C 180,E1 -18519.104,E2 -18519.104} C_VEL
LIN {X 0,Y 256.309,Z 361.371,A -85,B 0,C 180,E1 -18524.084,E2 -18524.084} C_VEL
LIN {X 0,Y 256.299,Z 361.372,A -85,B 0,C 180,E1 -18528.932,E2 -18528.932} C_VEL
LIN {X 0,Y 256.503,Z 361.347,A -85,B 0,C 180,E1 -18532.124,E2 -18532.124} C_VEL
LIN {X 0,Y 256.497,Z 361.348,A -85,B 0,C 180,E1 -18536.857,E2 -18536.857} C_VEL
LIN {X 0,Y 256.765,Z 361.316,A -85,B 0,C 180,E1 -18539.998,E2 -18539.998} C_VEL
LIN {X 0,Y 256.502,Z 361.345,A -85,B 0,C 180,E1 -18543.14,E2 -18543.14} C_VEL
LIN {X 0,Y 256.51,Z 361.346,A -85,B 0,C 180,E1 -18547.872,E2 -18547.872} C_VEL
LIN {X 0,Y 256.295,Z 361.374,A -85,B 0,C 180,E1 -18551.065,E2 -18551.065} C_VEL
LIN {X 0,Y 256.295,Z 361.671,A -85,B 0,C 180,E1 -18552.67,E2 -18552.67} C_VEL
LIN {X 0,Y 256.439,Z 363.793,A -85,B 0,C 180,E1 -18556.415,E2 -18556.415} C_VEL
LIN {X 0,Y 256.156,Z 366.676,A -85,B 0,C 180,E1 -18560.894,E2 -18560.894} C_VEL
LIN {X 0,Y 255.793,Z 369.261,A -85,B 0,C 180,E1 -18564.645,E2 -18564.645} C_VEL
LIN {X 0,Y 256.874,Z 372.538,A -85,B 0,C 180,E1 -18565.058,E2 -18565.058} C_VEL
LIN {X 0,Y 260.088,Z 381.453,A -85,B 0,C 180,E1 -18566.26,E2 -18566.26} C_VEL
LIN {X 0,Y 262.427,Z 390.426,A -85,B 0,C 180,E1 -18567.555,E2 -18567.555} C_VEL
LIN {X 0,Y 263.809,Z 397.338,A -85,B 0,C 180,E1 -18568.653,E2 -18568.653} C_VEL
LIN {X 0,Y 264.613,Z 404.35,A -85,B 0,C 180,E1 -18569.865,E2 -18569.865} C_VEL
LIN {X 0,Y 264.18,Z 408.206,A -85,B 0,C 180,E1 -18570.504,E2 -18570.504} C_VEL
LIN {X 0,Y 262.289,Z 416.769,A -85,B 0,C 180,E1 -18572.123,E2 -18572.123} C_VEL
LIN {X 0,Y 260.933,Z 422.981,A -85,B 0,C 180,E1 -18573.602,E2 -18573.602} C_VEL
LIN {X 0,Y 259.262,Z 429.667,A -85,B 0,C 180,E1 -18575.584,E2 -18575.584} C_VEL
LIN {X 0,Y 258.017,Z 434.188,A -85,B 0,C 180,E1 -18577.244,E2 -18577.244} C_VEL
LIN {X 0,Y 257.005,Z 437.977,A -85,B 0,C 180,E1 -18578.97,E2 -18578.97} C_VEL
LIN {X 0,Y 255.859,Z 441.752,A -85,B 0,C 180,E1 -18581.239,E2 -18581.239} C_VEL
LIN {X 0,Y 254.979,Z 444.394,A -85,B 0,C 180,E1 -18583.554,E2 -18583.554} C_VEL
LIN {X 0,Y 254.315,Z 446.077,A -85,B 0,C 180,E1 -18586.298,E2 -18586.298} C_VEL
LIN {X 0,Y 253.979,Z 446.315,A -85,B 0,C 180,E1 -18588.383,E2 -18588.383} C_VEL
LIN {X 0,Y 253.904,Z 445.469,A -85,B 0,C 180,E1 -18590.805,E2 -18590.805} C_VEL
LIN {X 0,Y 254.093,Z 443.361,A -85,B 0,C 180,E1 -18593.329,E2 -18593.329} C_VEL
LIN {X 0,Y 254.553,Z 439.847,A -85,B 0,C 180,E1 -18595.918,E2 -18595.918} C_VEL
LIN {X 0,Y 255.209,Z 434.709,A -85,B 0,C 180,E1 -18598.449,E2 -18598.449} C_VEL
LIN {X 0,Y 255.865,Z 429.622,A -85,B 0,C 180,E1 -18600.367,E2 -18600.367} C_VEL
LIN {X 0,Y 256.511,Z 425.028,A -85,B 0,C 180,E1 -18601.797,E2 -18601.797} C_VEL
LIN {X 0,Y 257.441,Z 417.677,A -85,B 0,C 180,E1 -18603.663,E2 -18603.663} C_VEL
LIN {X 0,Y 258.501,Z 409.715,A -85,B 0,C 180,E1 -18605.289,E2 -18605.289} C_VEL
LIN {X 0,Y 259.687,Z 399.438,A -85,B 0,C 180,E1 -18606.943,E2 -18606.943} C_VEL
LIN {X 0,Y 259.729,Z 395.101,A -85,B 0,C 180,E1 -18607.527,E2 -18607.527} C_VEL
LIN {X 0,Y 258.167,Z 384.803,A -85,B 0,C 180,E1 -18608.803,E2 -18608.803} C_VEL
LIN {X 0,Y 256.106,Z 373.737,A -85,B 0,C 180,E1 -18609.84,E2 -18609.84} C_VEL
LIN {X 0,Y 254.728,Z 367.106,A -85,B 0,C 180,E1 -18610.377,E2 -18610.377} C_VEL
LIN {X 0,Y 255.132,Z 362.516,A -85,B 0,C 180,E1 -18615.644,E2 -18615.644} C_VEL
LIN {X 0,Y 255.273,Z 361.504,A -85,B 0,C 180,E1 -18616.87,E2 -18616.87} C_VEL
LIN {X 0,Y 256.06,Z 361.4,A -85,B 0,C 180,E1 -18621.131,E2 -18621.131} C_VEL
LIN {X 0,Y 256.391,Z 361.36,A -85,B 0,C 180,E1 -18623.703,E2 -18623.703} C_VEL
LIN {X 0,Y 256.706,Z 361.322,A -85,B 0,C 180,E1 -18628.429,E2 -18628.429} C_VEL
LIN {X 0,Y 256.706,Z 361.321,A -85,B 0,C 180,E1 -18631.567,E2 -18631.567} C_VEL
LIN {X 0,Y 256.531,Z 361.345,A -85,B 0,C 180,E1 -18637.871,E2 -18637.871} C_VEL
LIN {X 0,Y 256.3,Z 361.368,A -85,B 0,C 180,E1 -18641.064,E2 -18641.064} C_VEL
LIN {X 0,Y 256.289,Z 361.374,A -85,B 0,C 180,E1 -18645.913,E2 -18645.913} C_VEL
LIN {X 0,Y 256.157,Z 361.386,A -85,B 0,C 180,E1 -18650.894,E2 -18650.894} C_VEL
LIN {X 0,Y 256.176,Z 361.387,A -85,B 0,C 180,E1 -18655.137,E2 -18655.137} C_VEL
LIN {X 0,Y 256.098,Z 361.397,A -85,B 0,C 180,E1 -18659.599,E2 -18659.599} C_VEL
LIN {X 0,Y 256.072,Z 361.402,A -85,B 0,C 180,E1 -18663.289,E2 -18663.289} C_VEL
LIN {X 0,Y 256.129,Z 361.393,A -85,B 0,C 180,E1 -18667.278,E2 -18667.278} C_VEL
LIN {X 0,Y 256.147,Z 361.392,A -85,B 0,C 180,E1 -18671.182,E2 -18671.182} C_VEL
LIN {X 0,Y 256.103,Z 361.394,A -85,B 0,C 180,E1 -18675.516,E2 -18675.516} C_VEL
LIN {X 0,Y 256.119,Z 361.395,A -85,B 0,C 180,E1 -18678.812,E2 -18678.812} C_VEL
LIN {X 0,Y 256.142,Z 361.391,A -85,B 0,C 180,E1 -18682.872,E2 -18682.872} C_VEL
LIN {X 0,Y 256.072,Z 361.402,A -85,B 0,C 180,E1 -18686.71,E2 -18686.71} C_VEL
LIN {X 0,Y 256.125,Z 361.389,A -85,B 0,C 180,E1 -18691.405,E2 -18691.405} C_VEL
LIN {X 0,Y 256.177,Z 361.385,A -85,B 0,C 180,E1 -18695.702,E2 -18695.702} C_VEL
LIN {X 0,Y 256.23,Z 361.376,A -85,B 0,C 180,E1 -18699.112,E2 -18699.112} C_VEL
LIN {X 0,Y 256.288,Z 361.373,A -85,B 0,C 180,E1 -18704.086,E2 -18704.086} C_VEL
LIN {X 0,Y 256.299,Z 361.369,A -85,B 0,C 180,E1 -18708.935,E2 -18708.935} C_VEL
LIN {X 0,Y 256.529,Z 361.345,A -85,B 0,C 180,E1 -18712.128,E2 -18712.128} C_VEL
LIN {X 0,Y 256.704,Z 361.32,A -85,B 0,C 180,E1 -18718.433,E2 -18718.433} C_VEL
LIN {X 0,Y 256.706,Z 361.321,A -85,B 0,C 180,E1 -18721.57,E2 -18721.57} C_VEL
LIN {X 0,Y 256.531,Z 361.344,A -85,B 0,C 180,E1 -18727.875,E2 -18727.875} C_VEL
LIN {X 0,Y 256.301,Z 361.369,A -85,B 0,C 180,E1 -18731.068,E2 -18731.068} C_VEL
LIN {X 0,Y 256.292,Z 361.372,A -85,B 0,C 180,E1 -18735.917,E2 -18735.917} C_VEL
LIN {X 0,Y 256.159,Z 361.386,A -85,B 0,C 180,E1 -18740.897,E2 -18740.897} C_VEL
LIN {X 0,Y 256.181,Z 361.387,A -85,B 0,C 180,E1 -18745.141,E2 -18745.141} C_VEL
LIN {X 0,Y 256.107,Z 361.394,A -85,B 0,C 180,E1 -18749.602,E2 -18749.602} C_VEL
LIN {X 0,Y 256.062,Z 361.402,A -85,B 0,C 180,E1 -18753.295,E2 -18753.295} C_VEL
LIN {X 0,Y 256.06,Z 361.398,A -85,B 0,C 180,E1 -18755.719,E2 -18755.719} C_VEL
LIN {X 0,Y 255.398,Z 361.484,A -85,B 0,C 180,E1 -18757.032,E2 -18757.032} C_VEL
LIN {X 0,Y 252.575,Z 361.836,A -85,B 0,C 180,E1 -18759.173,E2 -18759.173} C_VEL
LIN {X 0,Y 250.163,Z 362.138,A -85,B 0,C 180,E1 -18760.915,E2 -18760.915} C_VEL
LIN {X 0,Y 249.107,Z 362.266,A -85,B 0,C 180,E1 -18762.266,E2 -18762.266} C_VEL
LIN {X 0,Y 249.01,Z 362.28,A -85,B 0,C 180,E1 -18762.723,E2 -18762.723} C_VEL
LIN {X 0,Y 249.131,Z 362.347,A -85,B 0,C 180,E1 -18767.528,E2 -18767.528} C_VEL
LIN {X 0,Y 250.067,Z 367.215,A -85,B 0,C 180,E1 -18771.901,E2 -18771.901} C_VEL
LIN {X 0,Y 250.55,Z 370.165,A -85,B 0,C 180,E1 -18774.437,E2 -18774.437} C_VEL
LIN {X 0,Y 250.674,Z 371.912,A -85,B 0,C 180,E1 -18775.897,E2 -18775.897} C_VEL
LIN {X 0,Y 249.877,Z 376.569,A -85,B 0,C 180,E1 -18779.587,E2 -18779.587} C_VEL
LIN {X 0,Y 248.781,Z 382.298,A -85,B 0,C 180,E1 -18784.035,E2 -18784.035} C_VEL
LIN {X 0,Y 247.895,Z 389.052,A -85,B 0,C 180,E1 -18789.187,E2 -18789.187} C_VEL
LIN {X 0,Y 249.299,Z 401.51,A -85,B 0,C 180,E1 -18790.116,E2 -18790.116} C_VEL
LIN {X 0,Y 250.126,Z 411.661,A -85,B 0,C 180,E1 -18791.15,E2 -18791.15} C_VEL
LIN {X 0,Y 250.74,Z 421.078,A -85,B 0,C 180,E1 -18792.364,E2 -18792.364} C_VEL
LIN {X 0,Y 250.972,Z 429.781,A -85,B 0,C 180,E1 -18793.74,E2 -18793.74} C_VEL
LIN {X 0,Y 249.927,Z 438.222,A -85,B 0,C 180,E1 -18795.342,E2 -18795.342} C_VEL
LIN {X 0,Y 248.829,Z 446.467,A -85,B 0,C 180,E1 -18797.358,E2 -18797.358} C_VEL
LIN {X 0,Y 248.157,Z 451.858,A -85,B 0,C 180,E1 -18798.981,E2 -18798.981} C_VEL
LIN {X 0,Y 247.583,Z 457.317,A -85,B 0,C 180,E1 -18801.02,E2 -18801.02} C_VEL
LIN {X 0,Y 247.261,Z 460.858,A -85,B 0,C 180,E1 -18802.654,E2 -18802.654} C_VEL
LIN {X 0,Y 247.016,Z 464.899,A -85,B 0,C 180,E1 -18805.106,E2 -18805.106} C_VEL
LIN {X 0,Y 247.073,Z 466.863,A -85,B 0,C 180,E1 -18806.741,E2 -18806.741} C_VEL
LIN {X 0,Y 247.073,Z 468.296,A -85,B 0,C 180,E1 -18808.372,E2 -18808.372} C_VEL
LIN {X 0,Y 247.095,Z 469.197,A -85,B 0,C 180,E1 -18810.002,E2 -18810.002} C_VEL
LIN {X 0,Y 247.054,Z 469.492,A -85,B 0,C 180,E1 -18811.632,E2 -18811.632} C_VEL
LIN {X 0,Y 247.007,Z 469.303,A -85,B 0,C 180,E1 -18813.264,E2 -18813.264} C_VEL
LIN {X 0,Y 246.994,Z 468.468,A -85,B 0,C 180,E1 -18815.184,E2 -18815.184} C_VEL
LIN {X 0,Y 247.089,Z 467.529,A -85,B 0,C 180,E1 -18816.535,E2 -18816.535} C_VEL
LIN {X 0,Y 247.613,Z 464.745,A -85,B 0,C 180,E1 -18818.983,E2 -18818.983} C_VEL
LIN {X 0,Y 248.498,Z 460.73,A -85,B 0,C 180,E1 -18821.42,E2 -18821.42} C_VEL
LIN {X 0,Y 249.348,Z 457.308,A -85,B 0,C 180,E1 -18823.033,E2 -18823.033} C_VEL
LIN {X 0,Y 250.675,Z 452.02,A -85,B 0,C 180,E1 -18825.033,E2 -18825.033} C_VEL
LIN {X 0,Y 252.002,Z 446.878,A -85,B 0,C 180,E1 -18826.612,E2 -18826.612} C_VEL
LIN {X 0,Y 253.581,Z 440.732,A -85,B 0,C 180,E1 -18828.169,E2 -18828.169} C_VEL
LIN {X 0,Y 254.568,Z 435.365,A -85,B 0,C 180,E1 -18829.349,E2 -18829.349} C_VEL
LIN {X 0,Y 255.109,Z 428.249,A -85,B 0,C 180,E1 -18830.735,E2 -18830.735} C_VEL
LIN {X 0,Y 255.155,Z 420.537,A -85,B 0,C 180,E1 -18832.044,E2 -18832.044} C_VEL
LIN {X 0,Y 254.571,Z 412.561,A -85,B 0,C 180,E1 -18833.257,E2 -18833.257} C_VEL
LIN {X 0,Y 253.386,Z 403.954,A -85,B 0,C 180,E1 -18834.422,E2 -18834.422} C_VEL
LIN {X 0,Y 251.119,Z 393.794,A -85,B 0,C 180,E1 -18835.66,E2 -18835.66} C_VEL
LIN {X 0,Y 249.384,Z 387.439,A -85,B 0,C 180,E1 -18836.365,E2 -18836.365} C_VEL
LIN {X 0,Y 249.31,Z 386.88,A -85,B 0,C 180,E1 -18836.428,E2 -18836.428} C_VEL
LIN {X 0,Y 250.384,Z 382.126,A -85,B 0,C 180,E1 -18840.349,E2 -18840.349} C_VEL
LIN {X 0,Y 251.172,Z 379.111,A -85,B 0,C 180,E1 -18842.919,E2 -18842.919} C_VEL
LIN {X 0,Y 251.376,Z 377.902,A -85,B 0,C 180,E1 -18844,E2 -18844} C_VEL
LIN {X 0,Y 251.172,Z 374.806,A -85,B 0,C 180,E1 -18846.986,E2 -18846.986} C_VEL
LIN {X 0,Y 250.624,Z 371.24,A -85,B 0,C 180,E1 -18850.786,E2 -18850.786} C_VEL
LIN {X 0,Y 249.912,Z 367.399,A -85,B 0,C 180,E1 -18855.326,E2 -18855.326} C_VEL
LIN {X 0,Y 249.384,Z 364.27,A -85,B 0,C 180,E1 -18859.595,E2 -18859.595} C_VEL
LIN {X 0,Y 249.118,Z 362.596,A -85,B 0,C 180,E1 -18862.181,E2 -18862.181} C_VEL
LIN {X 0,Y 249.054,Z 362.275,A -85,B 0,C 180,E1 -18864.922,E2 -18864.922} C_VEL
LIN {X 0,Y 249.057,Z 362.274,A -85,B 0,C 180,E1 -18869.472,E2 -18869.472} C_VEL
LIN {X 0,Y 249.081,Z 362.273,A -85,B 0,C 180,E1 -18873.162,E2 -18873.162} C_VEL
LIN {X 0,Y 249.089,Z 362.27,A -85,B 0,C 180,E1 -18876.732,E2 -18876.732} C_VEL
LIN {X 0,Y 249.12,Z 362.266,A -85,B 0,C 180,E1 -18880.211,E2 -18880.211} C_VEL
LIN {X 0,Y 249.251,Z 362.251,A -85,B 0,C 180,E1 -18883.621,E2 -18883.621} C_VEL
LIN {X 0,Y 249.247,Z 362.251,A -85,B 0,C 180,E1 -18888.615,E2 -18888.615} C_VEL
LIN {X 0,Y 249.447,Z 362.226,A -85,B 0,C 180,E1 -18891.9,E2 -18891.9} C_VEL
LIN {X 0,Y 249.288,Z 362.246,A -85,B 0,C 180,E1 -18895.147,E2 -18895.147} C_VEL
LIN {X 0,Y 249.68,Z 362.193,A -85,B 0,C 180,E1 -18898.385,E2 -18898.385} C_VEL
LIN {X 0,Y 249.682,Z 362.194,A -85,B 0,C 180,E1 -18901.611,E2 -18901.611} C_VEL
LIN {X 0,Y 249.44,Z 362.227,A -85,B 0,C 180,E1 -18906.698,E2 -18906.698} C_VEL
LIN {X 0,Y 249.348,Z 362.24,A -85,B 0,C 180,E1 -18909.735,E2 -18909.735} C_VEL
LIN {X 0,Y 249.244,Z 362.355,A -85,B 0,C 180,E1 -18911.382,E2 -18911.382} C_VEL
LIN {X 0,Y 249.446,Z 364.096,A -85,B 0,C 180,E1 -18914.687,E2 -18914.687} C_VEL
LIN {X 0,Y 249.432,Z 365.227,A -85,B 0,C 180,E1 -18916.662,E2 -18916.662} C_VEL
LIN {X 0,Y 249.217,Z 367.137,A -85,B 0,C 180,E1 -18919.778,E2 -18919.778} C_VEL
LIN {X 0,Y 248.841,Z 369.693,A -85,B 0,C 180,E1 -18923.62,E2 -18923.62} C_VEL
LIN {X 0,Y 249.964,Z 372.867,A -85,B 0,C 180,E1 -18924.057,E2 -18924.057} C_VEL
LIN {X 0,Y 253.383,Z 382.254,A -85,B 0,C 180,E1 -18925.397,E2 -18925.397} C_VEL
LIN {X 0,Y 255.652,Z 390.346,A -85,B 0,C 180,E1 -18926.641,E2 -18926.641} C_VEL
LIN {X 0,Y 257.16,Z 398.054,A -85,B 0,C 180,E1 -18927.926,E2 -18927.926} C_VEL
LIN {X 0,Y 258.055,Z 405.895,A -85,B 0,C 180,E1 -18929.363,E2 -18929.363} C_VEL
LIN {X 0,Y 257.144,Z 411.554,A -85,B 0,C 180,E1 -18930.37,E2 -18930.37} C_VEL
LIN {X 0,Y 255.715,Z 417.515,A -85,B 0,C 180,E1 -18931.568,E2 -18931.568} C_VEL
LIN {X 0,Y 254.276,Z 423.666,A -85,B 0,C 180,E1 -18933.082,E2 -18933.082} C_VEL
LIN {X 0,Y 252.689,Z 429.592,A -85,B 0,C 180,E1 -18934.866,E2 -18934.866} C_VEL
LIN {X 0,Y 251.406,Z 434.067,A -85,B 0,C 180,E1 -18936.513,E2 -18936.513} C_VEL
LIN {X 0,Y 250.031,Z 438.777,A -85,B 0,C 180,E1 -18938.736,E2 -18938.736} C_VEL
LIN {X 0,Y 248.65,Z 443.069,A -85,B 0,C 180,E1 -18941.536,E2 -18941.536} C_VEL
LIN {X 0,Y 248.151,Z 444.366,A -85,B 0,C 180,E1 -18942.819,E2 -18942.819} C_VEL
LIN {X 0,Y 247.432,Z 446.07,A -85,B 0,C 180,E1 -18945.24,E2 -18945.24} C_VEL
LIN {X 0,Y 246.973,Z 446.688,A -85,B 0,C 180,E1 -18947.717,E2 -18947.717} C_VEL
LIN {X 0,Y 246.798,Z 446.076,A -85,B 0,C 180,E1 -18950.249,E2 -18950.249} C_VEL
LIN {X 0,Y 246.999,Z 443.661,A -85,B 0,C 180,E1 -18953.305,E2 -18953.305} C_VEL
LIN {X 0,Y 247.359,Z 440.844,A -85,B 0,C 180,E1 -18955.478,E2 -18955.478} C_VEL
LIN {X 0,Y 247.79,Z 437.481,A -85,B 0,C 180,E1 -18957.39,E2 -18957.39} C_VEL
LIN {X 0,Y 248.549,Z 431.922,A -85,B 0,C 180,E1 -18959.823,E2 -18959.823} C_VEL
LIN {X 0,Y 249.406,Z 425.858,A -85,B 0,C 180,E1 -18961.834,E2 -18961.834} C_VEL
LIN {X 0,Y 250.319,Z 419.028,A -85,B 0,C 180,E1 -18963.651,E2 -18963.651} C_VEL
LIN {X 0,Y 251.275,Z 411.937,A -85,B 0,C 180,E1 -18965.192,E2 -18965.192} C_VEL
LIN {X 0,Y 252.138,Z 404.879,A -85,B 0,C 180,E1 -18966.463,E2 -18966.463} C_VEL
LIN {X 0,Y 252.884,Z 396.963,A -85,B 0,C 180,E1 -18967.642,E2 -18967.642} C_VEL
LIN {X 0,Y 251.543,Z 387.958,A -85,B 0,C 180,E1 -18968.84,E2 -18968.84} C_VEL
LIN {X 0,Y 249.887,Z 378.276,A -85,B 0,C 180,E1 -18969.883,E2 -18969.883} C_VEL
LIN {X 0,Y 247.674,Z 367.435,A -85,B 0,C 180,E1 -18970.791,E2 -18970.791} C_VEL
LIN {X 0,Y 248.017,Z 363.656,A -85,B 0,C 180,E1 -18975.223,E2 -18975.223} C_VEL
LIN {X 0,Y 248.217,Z 362.382,A -85,B 0,C 180,E1 -18976.906,E2 -18976.906} C_VEL
LIN {X 0,Y 249.147,Z 362.263,A -85,B 0,C 180,E1 -18981.89,E2 -18981.89} C_VEL
LIN {X 0,Y 249.345,Z 362.237,A -85,B 0,C 180,E1 -18983.524,E2 -18983.524} C_VEL
LIN {X 0,Y 249.667,Z 362.199,A -85,B 0,C 180,E1 -18988.385,E2 -18988.385} C_VEL
LIN {X 0,Y 249.668,Z 362.198,A -85,B 0,C 180,E1 -18991.611,E2 -18991.611} C_VEL
LIN {X 0,Y 249.453,Z 362.223,A -85,B 0,C 180,E1 -18996.469,E2 -18996.469} C_VEL
LIN {X 0,Y 249.414,Z 362.23,A -85,B 0,C 180,E1 -18999.731,E2 -18999.731} C_VEL
LIN {X 0,Y 249.195,Z 362.254,A -85,B 0,C 180,E1 -19004.702,E2 -19004.702} C_VEL
LIN {X 0,Y 249.128,Z 362.263,A -85,B 0,C 180,E1 -19008.076,E2 -19008.076} C_VEL
LIN {X 0,Y 249.076,Z 362.271,A -85,B 0,C 180,E1 -19011.517,E2 -19011.517} C_VEL
LIN {X 0,Y 249.118,Z 362.268,A -85,B 0,C 180,E1 -19015.481,E2 -19015.481} C_VEL
LIN {X 0,Y 249.068,Z 362.27,A -85,B 0,C 180,E1 -19018.991,E2 -19018.991} C_VEL
LIN {X 0,Y 249.023,Z 362.276,A -85,B 0,C 180,E1 -19022.424,E2 -19022.424} C_VEL
LIN {X 0,Y 249.063,Z 362.269,A -85,B 0,C 180,E1 -19026.337,E2 -19026.337} C_VEL
LIN {X 0,Y 249.085,Z 362.269,A -85,B 0,C 180,E1 -19030.459,E2 -19030.459} C_VEL
LIN {X 0,Y 249.081,Z 362.271,A -85,B 0,C 180,E1 -19032.813,E2 -19032.813} C_VEL
LIN {X 0,Y 249.085,Z 362.27,A -85,B 0,C 180,E1 -19037.38,E2 -19037.38} C_VEL
LIN {X 0,Y 249.04,Z 362.273,A -85,B 0,C 180,E1 -19041.625,E2 -19041.625} C_VEL
LIN {X 0,Y 249.048,Z 362.273,A -85,B 0,C 180,E1 -19045.643,E2 -19045.643} C_VEL
LIN {X 0,Y 249.039,Z 362.273,A -85,B 0,C 180,E1 -19049.474,E2 -19049.474} C_VEL
LIN {X 0,Y 249.064,Z 362.271,A -85,B 0,C 180,E1 -19053.163,E2 -19053.163} C_VEL
LIN {X 0,Y 249.106,Z 362.268,A -85,B 0,C 180,E1 -19056.737,E2 -19056.737} C_VEL
LIN {X 0,Y 249.14,Z 362.262,A -85,B 0,C 180,E1 -19060.216,E2 -19060.216} C_VEL
LIN {X 0,Y 249.23,Z 362.25,A -85,B 0,C 180,E1 -19063.623,E2 -19063.623} C_VEL
LIN {X 0,Y 249.242,Z 362.249,A -85,B 0,C 180,E1 -19068.618,E2 -19068.618} C_VEL
LIN {X 0,Y 249.473,Z 362.222,A -85,B 0,C 180,E1 -19071.904,E2 -19071.904} C_VEL
LIN {X 0,Y 249.427,Z 362.224,A -85,B 0,C 180,E1 -19076.771,E2 -19076.771} C_VEL
LIN {X 0,Y 249.718,Z 362.193,A -85,B 0,C 180,E1 -19080.002,E2 -19080.002} C_VEL
LIN {X 0,Y 249.429,Z 362.225,A -85,B 0,C 180,E1 -19083.232,E2 -19083.232} C_VEL
LIN {X 0,Y 249.475,Z 362.222,A -85,B 0,C 180,E1 -19088.099,E2 -19088.099} C_VEL
LIN {X 0,Y 249.245,Z 362.25,A -85,B 0,C 180,E1 -19091.385,E2 -19091.385} C_VEL
LIN {X 0,Y 249.234,Z 362.25,A -85,B 0,C 180,E1 -19096.38,E2 -19096.38} C_VEL
LIN {X 0,Y 249.08,Z 362.271,A -85,B 0,C 180,E1 -19101.52,E2 -19101.52} C_VEL
LIN {X 0,Y 249.124,Z 362.266,A -85,B 0,C 180,E1 -19105.484,E2 -19105.484} C_VEL
LIN {X 0,Y 249.077,Z 362.27,A -85,B 0,C 180,E1 -19108.996,E2 -19108.996} C_VEL
LIN {X 0,Y 249.025,Z 362.276,A -85,B 0,C 180,E1 -19112.428,E2 -19112.428} C_VEL
LIN {X 0,Y 249.024,Z 362.275,A -85,B 0,C 180,E1 -19116.348,E2 -19116.348} C_VEL
LIN {X 0,Y 249.001,Z 362.279,A -85,B 0,C 180,E1 -19120.48,E2 -19120.48} C_VEL
LIN {X 0,Y 249.01,Z 362.28,A -85,B 0,C 180,E1 -19122.723,E2 -19122.723} C_VEL
LIN {X 0,Y 248.281,Z 362.419,A -85,B 0,C 180,E1 -19123.631,E2 -19123.631} C_VEL
LIN {X 0,Y 245.35,Z 362.734,A -85,B 0,C 180,E1 -19125.056,E2 -19125.056} C_VEL
LIN {X 0,Y 242.574,Z 363.08,A -85,B 0,C 180,E1 -19126.501,E2 -19126.501} C_VEL
LIN {X 0,Y 242.084,Z 363.301,A -85,B 0,C 180,E1 -19127.419,E2 -19127.419} C_VEL
LIN {X 0,Y 242.893,Z 367.562,A -85,B 0,C 180,E1 -19131.375,E2 -19131.375} C_VEL
LIN {X 0,Y 243.51,Z 371.355,A -85,B 0,C 180,E1 -19134.747,E2 -19134.747} C_VEL
LIN {X 0,Y 243.43,Z 373.857,A -85,B 0,C 180,E1 -19136.853,E2 -19136.853} C_VEL
LIN {X 0,Y 242.561,Z 378.35,A -85,B 0,C 180,E1 -19140.494,E2 -19140.494} C_VEL
LIN {X 0,Y 241.314,Z 385.195,A -85,B 0,C 180,E1 -19145.94,E2 -19145.94} C_VEL
LIN {X 0,Y 240.843,Z 388.834,A -85,B 0,C 180,E1 -19148.751,E2 -19148.751} C_VEL
LIN {X 0,Y 242.307,Z 401.706,A -85,B 0,C 180,E1 -19149.745,E2 -19149.745} C_VEL
LIN {X 0,Y 243.129,Z 411.692,A -85,B 0,C 180,E1 -19150.806,E2 -19150.806} C_VEL
LIN {X 0,Y 243.721,Z 421.367,A -85,B 0,C 180,E1 -19152.103,E2 -19152.103} C_VEL
LIN {X 0,Y 243.915,Z 430.922,A -85,B 0,C 180,E1 -19153.687,E2 -19153.687} C_VEL
LIN {X 0,Y 242.758,Z 438.977,A -85,B 0,C 180,E1 -19155.328,E2 -19155.328} C_VEL
LIN {X 0,Y 241.868,Z 445.568,A -85,B 0,C 180,E1 -19156.988,E2 -19156.988} C_VEL
LIN {X 0,Y 241.172,Z 451.058,A -85,B 0,C 180,E1 -19158.658,E2 -19158.658} C_VEL
LIN {X 0,Y 240.555,Z 456.603,A -85,B 0,C 180,E1 -19160.756,E2 -19160.756} C_VEL
LIN {X 0,Y 240.092,Z 461.741,A -85,B 0,C 180,E1 -19163.278,E2 -19163.278} C_VEL
LIN {X 0,Y 239.918,Z 465.111,A -85,B 0,C 180,E1 -19165.531,E2 -19165.531} C_VEL
LIN {X 0,Y 240.002,Z 467.866,A -85,B 0,C 180,E1 -19168.324,E2 -19168.324} C_VEL
LIN {X 0,Y 240.021,Z 468.781,A -85,B 0,C 180,E1 -19170.002,E2 -19170.002} C_VEL
LIN {X 0,Y 239.982,Z 469.123,A -85,B 0,C 180,E1 -19171.68,E2 -19171.68} C_VEL
LIN {X 0,Y 239.904,Z 468.994,A -85,B 0,C 180,E1 -19173.361,E2 -19173.361} C_VEL
LIN {X 0,Y 239.885,Z 468.405,A -85,B 0,C 180,E1 -19175.044,E2 -19175.044} C_VEL
LIN {X 0,Y 240.037,Z 467.33,A -85,B 0,C 180,E1 -19176.728,E2 -19176.728} C_VEL
LIN {X 0,Y 240.587,Z 464.648,A -85,B 0,C 180,E1 -19179.248,E2 -19179.248} C_VEL
LIN {X 0,Y 241.531,Z 460.72,A -85,B 0,C 180,E1 -19181.755,E2 -19181.755} C_VEL
LIN {X 0,Y 242.96,Z 455.441,A -85,B 0,C 180,E1 -19184.236,E2 -19184.236} C_VEL
LIN {X 0,Y 244.843,Z 448.559,A -85,B 0,C 180,E1 -19186.683,E2 -19186.683} C_VEL
LIN {X 0,Y 246.861,Z 441.118,A -85,B 0,C 180,E1 -19188.682,E2 -19188.682} C_VEL
LIN {X 0,Y 248.08,Z 434.288,A -85,B 0,C 180,E1 -19190.223,E2 -19190.223} C_VEL
LIN {X 0,Y 248.574,Z 426.421,A -85,B 0,C 180,E1 -19191.785,E2 -19191.785} C_VEL
LIN {X 0,Y 248.506,Z 418.809,A -85,B 0,C 180,E1 -19193.106,E2 -19193.106} C_VEL
LIN {X 0,Y 247.681,Z 409.519,A -85,B 0,C 180,E1 -19194.536,E2 -19194.536} C_VEL
LIN {X 0,Y 246.108,Z 400.77,A -85,B 0,C 180,E1 -19195.756,E2 -19195.756} C_VEL
LIN {X 0,Y 243.299,Z 389.645,A -85,B 0,C 180,E1 -19197.174,E2 -19197.174} C_VEL
LIN {X 0,Y 242.519,Z 386.497,A -85,B 0,C 180,E1 -19197.503,E2 -19197.503} C_VEL
LIN {X 0,Y 243.58,Z 382.095,A -85,B 0,C 180,E1 -19201.291,E2 -19201.291} C_VEL
LIN {X 0,Y 244.256,Z 379.683,A -85,B 0,C 180,E1 -19203.443,E2 -19203.443} C_VEL
LIN {X 0,Y 244.259,Z 376.715,A -85,B 0,C 180,E1 -19206.326,E2 -19206.326} C_VEL
LIN {X 0,Y 243.88,Z 373.901,A -85,B 0,C 180,E1 -19209.347,E2 -19209.347} C_VEL
LIN {X 0,Y 243.186,Z 370.139,A -85,B 0,C 180,E1 -19213.738,E2 -19213.738} C_VEL
LIN {X 0,Y 242.574,Z 366.798,A -85,B 0,C 180,E1 -19218.211,E2 -19218.211} C_VEL
LIN {X 0,Y 242.179,Z 364.063,A -85,B 0,C 180,E1 -19222.451,E2 -19222.451} C_VEL
LIN {X 0,Y 241.997,Z 363.154,A -85,B 0,C 180,E1 -19224.489,E2 -19224.489} C_VEL
LIN {X 0,Y 241.982,Z 363.155,A -85,B 0,C 180,E1 -19228.479,E2 -19228.479} C_VEL
LIN {X 0,Y 242.012,Z 363.152,A -85,B 0,C 180,E1 -19232.312,E2 -19232.312} C_VEL
LIN {X 0,Y 242.067,Z 363.146,A -85,B 0,C 180,E1 -19236.015,E2 -19236.015} C_VEL
LIN {X 0,Y 242.047,Z 363.147,A -85,B 0,C 180,E1 -19239.607,E2 -19239.607} C_VEL
LIN {X 0,Y 242.173,Z 363.131,A -85,B 0,C 180,E1 -19243.277,E2 -19243.277} C_VEL
LIN {X 0,Y 242.184,Z 363.132,A -85,B 0,C 180,E1 -19248.278,E2 -19248.278} C_VEL
LIN {X 0,Y 242.396,Z 363.105,A -85,B 0,C 180,E1 -19251.663,E2 -19251.663} C_VEL
LIN {X 0,Y 242.248,Z 363.122,A -85,B 0,C 180,E1 -19255.005,E2 -19255.005} C_VEL
LIN {X 0,Y 242.641,Z 363.07,A -85,B 0,C 180,E1 -19258.339,E2 -19258.339} C_VEL
LIN {X 0,Y 242.642,Z 363.071,A -85,B 0,C 180,E1 -19261.658,E2 -19261.658} C_VEL
LIN {X 0,Y 242.422,Z 363.103,A -85,B 0,C 180,E1 -19266.669,E2 -19266.669} C_VEL
LIN {X 0,Y 242.272,Z 363.12,A -85,B 0,C 180,E1 -19270.022,E2 -19270.022} C_VEL
LIN {X 0,Y 242.401,Z 364.736,A -85,B 0,C 180,E1 -19273.41,E2 -19273.41} C_VEL
LIN {X 0,Y 242.418,Z 366.657,A -85,B 0,C 180,E1 -19276.914,E2 -19276.914} C_VEL
LIN {X 0,Y 242.034,Z 369.565,A -85,B 0,C 180,E1 -19281.686,E2 -19281.686} C_VEL
LIN {X 0,Y 241.925,Z 370.205,A -85,B 0,C 180,E1 -19282.524,E2 -19282.524} C_VEL
LIN {X 0,Y 243.084,Z 373.396,A -85,B 0,C 180,E1 -19282.972,E2 -19282.972} C_VEL
LIN {X 0,Y 246.599,Z 382.588,A -85,B 0,C 180,E1 -19284.407,E2 -19284.407} C_VEL
LIN {X 0,Y 249.203,Z 391.833,A -85,B 0,C 180,E1 -19285.919,E2 -19285.919} C_VEL
LIN {X 0,Y 250.724,Z 399.754,A -85,B 0,C 180,E1 -19287.321,E2 -19287.321} C_VEL
LIN {X 0,Y 251.48,Z 406.676,A -85,B 0,C 180,E1 -19288.665,E2 -19288.665} C_VEL
LIN {X 0,Y 251.409,Z 409.162,A -85,B 0,C 180,E1 -19289.133,E2 -19289.133} C_VEL
LIN {X 0,Y 249.262,Z 417.893,A -85,B 0,C 180,E1 -19290.887,E2 -19290.887} C_VEL
LIN {X 0,Y 247.533,Z 424.732,A -85,B 0,C 180,E1 -19292.644,E2 -19292.644} C_VEL
LIN {X 0,Y 246.176,Z 429.52,A -85,B 0,C 180,E1 -19294.112,E2 -19294.112} C_VEL
LIN {X 0,Y 244.378,Z 435.359,A -85,B 0,C 180,E1 -19296.363,E2 -19296.363} C_VEL
LIN {X 0,Y 243.403,Z 438.632,A -85,B 0,C 180,E1 -19297.955,E2 -19297.955} C_VEL
LIN {X 0,Y 242.389,Z 441.46,A -85,B 0,C 180,E1 -19299.631,E2 -19299.631} C_VEL
LIN {X 0,Y 241.338,Z 444.368,A -85,B 0,C 180,E1 -19302.048,E2 -19302.048} C_VEL
LIN {X 0,Y 240.524,Z 446.21,A -85,B 0,C 180,E1 -19304.526,E2 -19304.526} C_VEL
LIN {X 0,Y 239.972,Z 446.974,A -85,B 0,C 180,E1 -19307.065,E2 -19307.065} C_VEL
LIN {X 0,Y 239.724,Z 446.546,A -85,B 0,C 180,E1 -19309.834,E2 -19309.834} C_VEL
LIN {X 0,Y 239.789,Z 444.932,A -85,B 0,C 180,E1 -19312.308,E2 -19312.308} C_VEL
LIN {X 0,Y 240.038,Z 443.037,A -85,B 0,C 180,E1 -19314.154,E2 -19314.154} C_VEL
LIN {X 0,Y 240.426,Z 440.006,A -85,B 0,C 180,E1 -19316.26,E2 -19316.26} C_VEL
LIN {X 0,Y 241.109,Z 434.867,A -85,B 0,C 180,E1 -19318.841,E2 -19318.841} C_VEL
LIN {X 0,Y 241.78,Z 430.165,A -85,B 0,C 180,E1 -19320.691,E2 -19320.691} C_VEL
LIN {X 0,Y 242.523,Z 424.957,A -85,B 0,C 180,E1 -19322.374,E2 -19322.374} C_VEL
LIN {X 0,Y 243.374,Z 418.902,A -85,B 0,C 180,E1 -19323.996,E2 -19323.996} C_VEL
LIN {X 0,Y 244.375,Z 411.723,A -85,B 0,C 180,E1 -19325.579,E2 -19325.579} C_VEL
LIN {X 0,Y 245.385,Z 403.683,A -85,B 0,C 180,E1 -19327.029,E2 -19327.029} C_VEL
LIN {X 0,Y 245.881,Z 397.487,A -85,B 0,C 180,E1 -19327.964,E2 -19327.964} C_VEL
LIN {X 0,Y 244.833,Z 390.336,A -85,B 0,C 180,E1 -19328.97,E2 -19328.97} C_VEL
LIN {X 0,Y 243.434,Z 382.056,A -85,B 0,C 180,E1 -19329.948,E2 -19329.948} C_VEL
LIN {X 0,Y 241.641,Z 372.593,A -85,B 0,C 180,E1 -19330.844,E2 -19330.844} C_VEL
LIN {X 0,Y 240.63,Z 367.741,A -85,B 0,C 180,E1 -19331.258,E2 -19331.258} C_VEL
LIN {X 0,Y 240.924,Z 364.805,A -85,B 0,C 180,E1 -19334.777,E2 -19334.777} C_VEL
LIN {X 0,Y 241.124,Z 363.267,A -85,B 0,C 180,E1 -19336.728,E2 -19336.728} C_VEL
LIN {X 0,Y 242.047,Z 363.146,A -85,B 0,C 180,E1 -19341.65,E2 -19341.65} C_VEL
LIN {X 0,Y 242.274,Z 363.118,A -85,B 0,C 180,E1 -19343.335,E2 -19343.335} C_VEL
LIN {X 0,Y 242.627,Z 363.077,A -85,B 0,C 180,E1 -19348.338,E2 -19348.338} C_VEL
LIN {X 0,Y 242.628,Z 363.075,A -85,B 0,C 180,E1 -19351.658,E2 -19351.658} C_VEL
LIN {X 0,Y 242.425,Z 363.098,A -85,B 0,C 180,E1 -19356.657,E2 -19356.657} C_VEL
LIN {X 0,Y 242.335,Z 363.11,A -85,B 0,C 180,E1 -19360.019,E2 -19360.019} C_VEL
LIN {X 0,Y 242.156,Z 363.132,A -85,B 0,C 180,E1 -19365.139,E2 -19365.139} C_VEL
LIN {X 0,Y 242.062,Z 363.142,A -85,B 0,C 180,E1 -19368.623,E2 -19368.623} C_VEL
LIN {X 0,Y 242.002,Z 363.151,A -85,B 0,C 180,E1 -19372.178,E2 -19372.178} C_VEL
LIN {X 0,Y 242.055,Z 363.145,A -85,B 0,C 180,E1 -19375.837,E2 -19375.837} C_VEL
LIN {X 0,Y 242.017,Z 363.151,A -85,B 0,C 180,E1 -19379.579,E2 -19379.579} C_VEL
LIN {X 0,Y 241.978,Z 363.156,A -85,B 0,C 180,E1 -19383.49,E2 -19383.49} C_VEL
LIN {X 0,Y 242.007,Z 363.151,A -85,B 0,C 180,E1 -19387.576,E2 -19387.576} C_VEL
LIN {X 0,Y 242.028,Z 363.147,A -85,B 0,C 180,E1 -19391.9,E2 -19391.9} C_VEL
LIN {X 0,Y 242.011,Z 363.149,A -85,B 0,C 180,E1 -19396.548,E2 -19396.548} C_VEL
LIN {X 0,Y 241.998,Z 363.152,A -85,B 0,C 180,E1 -19400.292,E2 -19400.292} C_VEL
LIN {X 0,Y 242.024,Z 363.148,A -85,B 0,C 180,E1 -19404.498,E2 -19404.498} C_VEL
LIN {X 0,Y 241.963,Z 363.158,A -85,B 0,C 180,E1 -19408.481,E2 -19408.481} C_VEL
LIN {X 0,Y 241.998,Z 363.151,A -85,B 0,C 180,E1 -19412.314,E2 -19412.314} C_VEL
LIN {X 0,Y 242.069,Z 363.143,A -85,B 0,C 180,E1 -19416.019,E2 -19416.019} C_VEL
LIN {X 0,Y 242.074,Z 363.139,A -85,B 0,C 180,E1 -19419.613,E2 -19419.613} C_VEL
LIN {X 0,Y 242.152,Z 363.132,A -85,B 0,C 180,E1 -19423.279,E2 -19423.279} C_VEL
LIN {X 0,Y 242.175,Z 363.131,A -85,B 0,C 180,E1 -19428.281,E2 -19428.281} C_VEL
LIN {X 0,Y 242.424,Z 363.099,A -85,B 0,C 180,E1 -19431.667,E2 -19431.667} C_VEL
LIN {X 0,Y 242.251,Z 363.118,A -85,B 0,C 180,E1 -19435.009,E2 -19435.009} C_VEL
LIN {X 0,Y 242.626,Z 363.074,A -85,B 0,C 180,E1 -19438.342,E2 -19438.342} C_VEL
LIN {X 0,Y 242.628,Z 363.075,A -85,B 0,C 180,E1 -19441.661,E2 -19441.661} C_VEL
LIN {X 0,Y 242.425,Z 363.098,A -85,B 0,C 180,E1 -19446.661,E2 -19446.661} C_VEL
LIN {X 0,Y 242.337,Z 363.11,A -85,B 0,C 180,E1 -19450.022,E2 -19450.022} C_VEL
LIN {X 0,Y 242.159,Z 363.132,A -85,B 0,C 180,E1 -19455.143,E2 -19455.143} C_VEL
LIN {X 0,Y 242.065,Z 363.142,A -85,B 0,C 180,E1 -19458.626,E2 -19458.626} C_VEL
LIN {X 0,Y 242.006,Z 363.149,A -85,B 0,C 180,E1 -19462.182,E2 -19462.182} C_VEL
LIN {X 0,Y 242.06,Z 363.144,A -85,B 0,C 180,E1 -19465.84,E2 -19465.84} C_VEL
LIN {X 0,Y 242.024,Z 363.148,A -85,B 0,C 180,E1 -19469.582,E2 -19469.582} C_VEL
LIN {X 0,Y 241.975,Z 363.156,A -85,B 0,C 180,E1 -19473.495,E2 -19473.495} C_VEL
LIN {X 0,Y 241.981,Z 363.152,A -85,B 0,C 180,E1 -19477.585,E2 -19477.585} C_VEL
LIN {X 0,Y 241.935,Z 363.159,A -85,B 0,C 180,E1 -19481.925,E2 -19481.925} C_VEL
LIN {X 0,Y 242.087,Z 363.215,A -85,B 0,C 180,E1 -19487.34,E2 -19487.34} C_VEL
LIN {X 0,Y 242.084,Z 363.301,A -85,B 0,C 180,E1 -19487.419,E2 -19487.419} C_VEL
LIN {X 0,Y 241.811,Z 364.813,A -85,B 0,C 180,E1 -19488.765,E2 -19488.765} C_VEL
LIN {X 0,Y 240.588,Z 366.442,A -85,B 0,C 180,E1 -19490.089,E2 -19490.089} C_VEL
LIN {X 0,Y 236.705,Z 370.913,A -85,B 0,C 180,E1 -19493.662,E2 -19493.662} C_VEL
LIN {X 0,Y 236.457,Z 371.989,A -85,B 0,C 180,E1 -19494.592,E2 -19494.592} C_VEL
LIN {X 0,Y 236.431,Z 373.994,A -85,B 0,C 180,E1 -19496.339,E2 -19496.339} C_VEL
LIN {X 0,Y 235.613,Z 378.222,A -85,B 0,C 180,E1 -19499.888,E2 -19499.888} C_VEL
LIN {X 0,Y 234.349,Z 384.643,A -85,B 0,C 180,E1 -19505.177,E2 -19505.177} C_VEL
LIN {X 0,Y 233.85,Z 388.421,A -85,B 0,C 180,E1 -19508.25,E2 -19508.25} C_VEL
LIN {X 0,Y 235.293,Z 401.721,A -85,B 0,C 180,E1 -19509.342,E2 -19509.342} C_VEL
LIN {X 0,Y 236.008,Z 409.777,A -85,B 0,C 180,E1 -19510.203,E2 -19510.203} C_VEL
LIN {X 0,Y 236.551,Z 418.618,A -85,B 0,C 180,E1 -19511.37,E2 -19511.37} C_VEL
LIN {X 0,Y 236.872,Z 427.101,A -85,B 0,C 180,E1 -19512.743,E2 -19512.743} C_VEL
LIN {X 0,Y 236.764,Z 431.904,A -85,B 0,C 180,E1 -19513.623,E2 -19513.623} C_VEL
LIN {X 0,Y 235.596,Z 439.668,A -85,B 0,C 180,E1 -19515.314,E2 -19515.314} C_VEL
LIN {X 0,Y 234.727,Z 446.092,A -85,B 0,C 180,E1 -19517.025,E2 -19517.025} C_VEL
LIN {X 0,Y 234.012,Z 451.432,A -85,B 0,C 180,E1 -19518.745,E2 -19518.745} C_VEL
LIN {X 0,Y 233.519,Z 455.887,A -85,B 0,C 180,E1 -19520.474,E2 -19520.474} C_VEL
LIN {X 0,Y 233.042,Z 461.102,A -85,B 0,C 180,E1 -19523.074,E2 -19523.074} C_VEL
LIN {X 0,Y 232.884,Z 463.768,A -85,B 0,C 180,E1 -19524.808,E2 -19524.808} C_VEL
LIN {X 0,Y 232.898,Z 465.866,A -85,B 0,C 180,E1 -19526.542,E2 -19526.542} C_VEL
LIN {X 0,Y 232.932,Z 467.415,A -85,B 0,C 180,E1 -19528.273,E2 -19528.273} C_VEL
LIN {X 0,Y 232.949,Z 468.344,A -85,B 0,C 180,E1 -19530.002,E2 -19530.002} C_VEL
LIN {X 0,Y 232.909,Z 468.751,A -85,B 0,C 180,E1 -19531.731,E2 -19531.731} C_VEL
LIN {X 0,Y 232.802,Z 468.296,A -85,B 0,C 180,E1 -19534.966,E2 -19534.966} C_VEL
LIN {X 0,Y 232.983,Z 467.117,A -85,B 0,C 180,E1 -19536.932,E2 -19536.932} C_VEL
LIN {X 0,Y 233.552,Z 464.558,A -85,B 0,C 180,E1 -19539.529,E2 -19539.529} C_VEL
LIN {X 0,Y 234.556,Z 460.709,A -85,B 0,C 180,E1 -19542.109,E2 -19542.109} C_VEL
LIN {X 0,Y 236.082,Z 455.513,A -85,B 0,C 180,E1 -19544.66,E2 -19544.66} C_VEL
LIN {X 0,Y 237.68,Z 450.004,A -85,B 0,C 180,E1 -19546.758,E2 -19546.758} C_VEL
LIN {X 0,Y 240.164,Z 441.573,A -85,B 0,C 180,E1 -19549.223,E2 -19549.223} C_VEL
LIN {X 0,Y 241.407,Z 435.087,A -85,B 0,C 180,E1 -19550.775,E2 -19550.775} C_VEL
LIN {X 0,Y 242.006,Z 427.266,A -85,B 0,C 180,E1 -19552.407,E2 -19552.407} C_VEL
LIN {X 0,Y 242.014,Z 419.902,A -85,B 0,C 180,E1 -19553.763,E2 -19553.763} C_VEL
LIN {X 0,Y 241.305,Z 410.835,A -85,B 0,C 180,E1 -19555.247,E2 -19555.247} C_VEL
LIN {X 0,Y 239.888,Z 402.272,A -85,B 0,C 180,E1 -19556.538,E2 -19556.538} C_VEL
LIN {X 0,Y 237.686,Z 393.012,A -85,B 0,C 180,E1 -19557.816,E2 -19557.816} C_VEL
LIN {X 0,Y 235.856,Z 386.626,A -85,B 0,C 180,E1 -19558.635,E2 -19558.635} C_VEL
LIN {X 0,Y 235.788,Z 386.054,A -85,B 0,C 180,E1 -19558.729,E2 -19558.729} C_VEL
LIN {X 0,Y 236.837,Z 382.101,A -85,B 0,C 180,E1 -19562.288,E2 -19562.288} C_VEL
LIN {X 0,Y 237.261,Z 380.013,A -85,B 0,C 180,E1 -19564.252,E2 -19564.252} C_VEL
LIN {X 0,Y 237.215,Z 377.466,A -85,B 0,C 180,E1 -19566.875,E2 -19566.875} C_VEL
LIN {X 0,Y 236.663,Z 373.966,A -85,B 0,C 180,E1 -19570.795,E2 -19570.795} C_VEL
LIN {X 0,Y 235.975,Z 370.157,A -85,B 0,C 180,E1 -19575.628,E2 -19575.628} C_VEL
LIN {X 0,Y 235.578,Z 367.838,A -85,B 0,C 180,E1 -19578.978,E2 -19578.978} C_VEL
LIN {X 0,Y 235.397,Z 366.445,A -85,B 0,C 180,E1 -19581.171,E2 -19581.171} C_VEL
LIN {X 0,Y 234.94,Z 364.144,A -85,B 0,C 180,E1 -19585.362,E2 -19585.362} C_VEL
LIN {X 0,Y 234.931,Z 364.034,A -85,B 0,C 180,E1 -19589.431,E2 -19589.431} C_VEL
LIN {X 0,Y 235.003,Z 364.025,A -85,B 0,C 180,E1 -19593.794,E2 -19593.794} C_VEL
LIN {X 0,Y 235.021,Z 364.023,A -85,B 0,C 180,E1 -19598.969,E2 -19598.969} C_VEL
LIN {X 0,Y 235.106,Z 364.011,A -85,B 0,C 180,E1 -19603.059,E2 -19603.059} C_VEL
LIN {X 0,Y 235.118,Z 364.01,A -85,B 0,C 180,E1 -19607.921,E2 -19607.921} C_VEL
LIN {X 0,Y 235.33,Z 363.985,A -85,B 0,C 180,E1 -19611.411,E2 -19611.411} C_VEL
LIN {X 0,Y 235.366,Z 363.98,A -85,B 0,C 180,E1 -19613.139,E2 -19613.139} C_VEL
LIN {X 0,Y 235.6,Z 363.947,A -85,B 0,C 180,E1 -19618.289,E2 -19618.289} C_VEL
LIN {X 0,Y 235.602,Z 363.948,A -85,B 0,C 180,E1 -19621.708,E2 -19621.708} C_VEL
LIN {X 0,Y 235.373,Z 363.98,A -85,B 0,C 180,E1 -19626.858,E2 -19626.858} C_VEL
LIN {X 0,Y 235.332,Z 363.985,A -85,B 0,C 180,E1 -19628.586,E2 -19628.586} C_VEL
LIN {X 0,Y 235.356,Z 365.449,A -85,B 0,C 180,E1 -19632.064,E2 -19632.064} C_VEL
LIN {X 0,Y 235.444,Z 367.227,A -85,B 0,C 180,E1 -19635.582,E2 -19635.582} C_VEL
